(* Logix 5000 project; controller reports 1756-L63 rev 20.15; software revision 20.04; part 16 of 52 *)

        [783].log_data[6].valid := 1, [783].log_data[7].valid := 1, [783].log_data[8].valid := 1, [783].log_data[9].valid := 1, [783].log_data[10].valid := 1, [783].log_data[11].valid := 1, [783].log_data[12].valid := 1, [783].log_data[13].valid := 1, [783].log_data[14].valid := 1, [783].log_data[15].valid := 1, [783].log_data[16].valid := 1, [783].log_data[17].valid := 1, [783].log_data[18].valid := 1, [783].log_data[19].valid := 1, [783].time.Year := 2023, [783].time.Month := 1, [783].time.Day := 12, [783].time.Hour := 9, [783].time.Minute := 39, [783].time.Second := 59, [784].log_data[0].min := 1.0, [784].log_data[0].max := 1.0, [784].log_data[0].total := 300.0, [784].log_data[0].time := 300.0, [784].log_data[0].minminute := 40, [784].log_data[0].maxminute := 40, [784].log_data[0].valid := 1, [784].log_data[1].valid := 1, [784].log_data[2].valid := 1, [784].log_data[3].valid := 1, [784].log_data[4].valid := 1, [784].log_data[5].valid := 1, [784].log_data[6].valid := 1, [784].log_data[7].valid := 1, [784].log_data[8].valid := 1, [784].log_data[9].valid := 1, [784].log_data[10].valid := 1, [784].log_data[11].valid := 1, [784].log_data[12].valid := 1, [784].log_data[13].valid := 1, [784].log_data[14].valid := 1, [784].log_data[15].valid := 1, [784].log_data[16].valid := 1, [784].log_data[17].valid := 1, [784].log_data[18].valid := 1, [784].log_data[19].valid := 1, [784].time.Year := 2023, [784].time.Month := 1, [784].time.Day := 12, [784].time.Hour := 9, [784].time.Minute := 44, [784].time.Second := 59, [785].log_data[0].min := 1.0, [785].log_data[0].max := 1.0, [785].log_data[0].total := 300.0, [785].log_data[0].time := 300.0, [785].log_data[0].minminute := 45, [785].log_data[0].maxminute := 45, [785].log_data[0].valid := 1, [785].log_data[1].valid := 1,
        [785].log_data[2].valid := 1, [785].log_data[3].valid := 1, [785].log_data[4].valid := 1, [785].log_data[5].valid := 1, [785].log_data[6].valid := 1, [785].log_data[7].valid := 1, [785].log_data[8].valid := 1, [785].log_data[9].valid := 1, [785].log_data[10].valid := 1, [785].log_data[11].valid := 1, [785].log_data[12].valid := 1, [785].log_data[13].valid := 1, [785].log_data[14].valid := 1, [785].log_data[15].valid := 1, [785].log_data[16].valid := 1, [785].log_data[17].valid := 1, [785].log_data[18].valid := 1, [785].log_data[19].valid := 1, [785].time.Year := 2023, [785].time.Month := 1, [785].time.Day := 12, [785].time.Hour := 9, [785].time.Minute := 49, [785].time.Second := 59, [786].log_data[0].min := 1.0, [786].log_data[0].max := 1.0, [786].log_data[0].total := 300.0, [786].log_data[0].time := 300.0, [786].log_data[0].minminute := 50, [786].log_data[0].maxminute := 50, [786].log_data[0].valid := 1, [786].log_data[1].valid := 1, [786].log_data[2].valid := 1, [786].log_data[3].valid := 1, [786].log_data[4].valid := 1, [786].log_data[5].valid := 1, [786].log_data[6].valid := 1, [786].log_data[7].valid := 1, [786].log_data[8].valid := 1, [786].log_data[9].valid := 1, [786].log_data[10].valid := 1, [786].log_data[11].valid := 1, [786].log_data[12].valid := 1, [786].log_data[13].valid := 1, [786].log_data[14].valid := 1, [786].log_data[15].valid := 1, [786].log_data[16].valid := 1, [786].log_data[17].valid := 1, [786].log_data[18].valid := 1, [786].log_data[19].valid := 1, [786].time.Year := 2023, [786].time.Month := 1, [786].time.Day := 12, [786].time.Hour := 9, [786].time.Minute := 54, [786].time.Second := 59, [787].log_data[0].min := 1.0, [787].log_data[0].max := 1.0, [787].log_data[0].total := 300.0, [787].log_data[0].time := 300.0,
        [787].log_data[0].minminute := 55, [787].log_data[0].maxminute := 55, [787].log_data[0].valid := 1, [787].log_data[1].valid := 1, [787].log_data[2].valid := 1, [787].log_data[3].valid := 1, [787].log_data[4].valid := 1, [787].log_data[5].valid := 1, [787].log_data[6].valid := 1, [787].log_data[7].valid := 1, [787].log_data[8].valid := 1, [787].log_data[9].valid := 1, [787].log_data[10].valid := 1, [787].log_data[11].valid := 1, [787].log_data[12].valid := 1, [787].log_data[13].valid := 1, [787].log_data[14].valid := 1, [787].log_data[15].valid := 1, [787].log_data[16].valid := 1, [787].log_data[17].valid := 1, [787].log_data[18].valid := 1, [787].log_data[19].valid := 1, [787].time.Year := 2023, [787].time.Month := 1, [787].time.Day := 12, [787].time.Hour := 9, [787].time.Minute := 59, [787].time.Second := 59, [788].log_data[0].min := 1.0, [788].log_data[0].max := 1.0, [788].log_data[0].total := 300.0, [788].log_data[0].time := 300.0, [788].log_data[0].valid := 1, [788].log_data[1].valid := 1, [788].log_data[2].valid := 1, [788].log_data[3].valid := 1, [788].log_data[4].valid := 1, [788].log_data[5].valid := 1, [788].log_data[6].valid := 1, [788].log_data[7].valid := 1, [788].log_data[8].valid := 1, [788].log_data[9].valid := 1, [788].log_data[10].valid := 1, [788].log_data[11].valid := 1, [788].log_data[12].valid := 1, [788].log_data[13].valid := 1, [788].log_data[14].valid := 1, [788].log_data[15].valid := 1, [788].log_data[16].valid := 1, [788].log_data[17].valid := 1, [788].log_data[18].valid := 1, [788].log_data[19].valid := 1, [788].time.Year := 2023, [788].time.Month := 1, [788].time.Day := 12, [788].time.Hour := 10, [788].time.Minute := 4, [788].time.Second := 59, [789].log_data[0].min := 1.0, [789].log_data[0].max := 1.0,
        [789].log_data[0].total := 300.0, [789].log_data[0].time := 300.0, [789].log_data[0].minminute := 5, [789].log_data[0].maxminute := 5, [789].log_data[0].valid := 1, [789].log_data[1].valid := 1, [789].log_data[2].valid := 1, [789].log_data[3].valid := 1, [789].log_data[4].valid := 1, [789].log_data[5].valid := 1, [789].log_data[6].valid := 1, [789].log_data[7].valid := 1, [789].log_data[8].valid := 1, [789].log_data[9].valid := 1, [789].log_data[10].valid := 1, [789].log_data[11].valid := 1, [789].log_data[12].valid := 1, [789].log_data[13].valid := 1, [789].log_data[14].valid := 1, [789].log_data[15].valid := 1, [789].log_data[16].valid := 1, [789].log_data[17].valid := 1, [789].log_data[18].valid := 1, [789].log_data[19].valid := 1, [789].time.Year := 2023, [789].time.Month := 1, [789].time.Day := 12, [789].time.Hour := 10, [789].time.Minute := 9, [789].time.Second := 59, [790].log_data[0].min := 1.0, [790].log_data[0].max := 1.0, [790].log_data[0].total := 300.0, [790].log_data[0].time := 300.0, [790].log_data[0].minminute := 10, [790].log_data[0].maxminute := 10, [790].log_data[0].valid := 1, [790].log_data[1].valid := 1, [790].log_data[2].valid := 1, [790].log_data[3].valid := 1, [790].log_data[4].valid := 1, [790].log_data[5].valid := 1, [790].log_data[6].valid := 1, [790].log_data[7].valid := 1, [790].log_data[8].valid := 1, [790].log_data[9].valid := 1, [790].log_data[10].valid := 1, [790].log_data[11].valid := 1, [790].log_data[12].valid := 1, [790].log_data[13].valid := 1, [790].log_data[14].valid := 1, [790].log_data[15].valid := 1, [790].log_data[16].valid := 1, [790].log_data[17].valid := 1, [790].log_data[18].valid := 1, [790].log_data[19].valid := 1, [790].time.Year := 2023, [790].time.Month := 1, [790].time.Day := 12, [790].time.Hour := 10,
        [790].time.Minute := 14, [790].time.Second := 59, [791].log_data[0].min := 1.0, [791].log_data[0].max := 1.0, [791].log_data[0].total := 300.0, [791].log_data[0].time := 300.0, [791].log_data[0].minminute := 15, [791].log_data[0].maxminute := 15, [791].log_data[0].valid := 1, [791].log_data[1].valid := 1, [791].log_data[2].valid := 1, [791].log_data[3].valid := 1, [791].log_data[4].valid := 1, [791].log_data[5].valid := 1, [791].log_data[6].valid := 1, [791].log_data[7].valid := 1, [791].log_data[8].valid := 1, [791].log_data[9].valid := 1, [791].log_data[10].valid := 1, [791].log_data[11].valid := 1, [791].log_data[12].valid := 1, [791].log_data[13].valid := 1, [791].log_data[14].valid := 1, [791].log_data[15].valid := 1, [791].log_data[16].valid := 1, [791].log_data[17].valid := 1, [791].log_data[18].valid := 1, [791].log_data[19].valid := 1, [791].time.Year := 2023, [791].time.Month := 1, [791].time.Day := 12, [791].time.Hour := 10, [791].time.Minute := 19, [791].time.Second := 59, [792].log_data[0].min := 1.0, [792].log_data[0].max := 1.0, [792].log_data[0].total := 300.0, [792].log_data[0].time := 300.0, [792].log_data[0].minminute := 20, [792].log_data[0].maxminute := 20, [792].log_data[0].valid := 1, [792].log_data[1].valid := 1, [792].log_data[2].valid := 1, [792].log_data[3].valid := 1, [792].log_data[4].valid := 1, [792].log_data[5].valid := 1, [792].log_data[6].valid := 1, [792].log_data[7].valid := 1, [792].log_data[8].valid := 1, [792].log_data[9].valid := 1, [792].log_data[10].valid := 1, [792].log_data[11].valid := 1, [792].log_data[12].valid := 1, [792].log_data[13].valid := 1, [792].log_data[14].valid := 1, [792].log_data[15].valid := 1, [792].log_data[16].valid := 1, [792].log_data[17].valid := 1, [792].log_data[18].valid := 1, [792].log_data[19].valid := 1,
        [792].time.Year := 2023, [792].time.Month := 1, [792].time.Day := 12, [792].time.Hour := 10, [792].time.Minute := 24, [792].time.Second := 59, [793].log_data[0].min := 1.0, [793].log_data[0].max := 1.0, [793].log_data[0].total := 300.0, [793].log_data[0].time := 300.0, [793].log_data[0].minminute := 25, [793].log_data[0].maxminute := 25, [793].log_data[0].valid := 1, [793].log_data[1].valid := 1, [793].log_data[2].valid := 1, [793].log_data[3].valid := 1, [793].log_data[4].valid := 1, [793].log_data[5].valid := 1, [793].log_data[6].valid := 1, [793].log_data[7].valid := 1, [793].log_data[8].valid := 1, [793].log_data[9].valid := 1, [793].log_data[10].valid := 1, [793].log_data[11].valid := 1, [793].log_data[12].valid := 1, [793].log_data[13].valid := 1, [793].log_data[14].valid := 1, [793].log_data[15].valid := 1, [793].log_data[16].valid := 1, [793].log_data[17].valid := 1, [793].log_data[18].valid := 1, [793].log_data[19].valid := 1, [793].time.Year := 2023, [793].time.Month := 1, [793].time.Day := 12, [793].time.Hour := 10, [793].time.Minute := 29, [793].time.Second := 59, [794].log_data[0].min := 1.0, [794].log_data[0].max := 1.0, [794].log_data[0].total := 300.0, [794].log_data[0].time := 300.0, [794].log_data[0].minminute := 30, [794].log_data[0].maxminute := 30, [794].log_data[0].valid := 1, [794].log_data[1].valid := 1, [794].log_data[2].valid := 1, [794].log_data[3].valid := 1, [794].log_data[4].valid := 1, [794].log_data[5].valid := 1, [794].log_data[6].valid := 1, [794].log_data[7].valid := 1, [794].log_data[8].valid := 1, [794].log_data[9].valid := 1, [794].log_data[10].valid := 1, [794].log_data[11].valid := 1, [794].log_data[12].valid := 1, [794].log_data[13].valid := 1, [794].log_data[14].valid := 1, [794].log_data[15].valid := 1,
        [794].log_data[16].valid := 1, [794].log_data[17].valid := 1, [794].log_data[18].valid := 1, [794].log_data[19].valid := 1, [794].time.Year := 2023, [794].time.Month := 1, [794].time.Day := 12, [794].time.Hour := 10, [794].time.Minute := 34, [794].time.Second := 59, [795].log_data[0].min := 1.0, [795].log_data[0].max := 1.0, [795].log_data[0].total := 300.0, [795].log_data[0].time := 300.0, [795].log_data[0].minminute := 35, [795].log_data[0].maxminute := 35, [795].log_data[0].valid := 1, [795].log_data[1].valid := 1, [795].log_data[2].valid := 1, [795].log_data[3].valid := 1, [795].log_data[4].valid := 1, [795].log_data[5].valid := 1, [795].log_data[6].valid := 1, [795].log_data[7].valid := 1, [795].log_data[8].valid := 1, [795].log_data[9].valid := 1, [795].log_data[10].valid := 1, [795].log_data[11].valid := 1, [795].log_data[12].valid := 1, [795].log_data[13].valid := 1, [795].log_data[14].valid := 1, [795].log_data[15].valid := 1, [795].log_data[16].valid := 1, [795].log_data[17].valid := 1, [795].log_data[18].valid := 1, [795].log_data[19].valid := 1, [795].time.Year := 2023, [795].time.Month := 1, [795].time.Day := 12, [795].time.Hour := 10, [795].time.Minute := 39, [795].time.Second := 59, [796].log_data[0].min := 1.0, [796].log_data[0].max := 1.0, [796].log_data[0].total := 300.0, [796].log_data[0].time := 300.0, [796].log_data[0].minminute := 40, [796].log_data[0].maxminute := 40, [796].log_data[0].valid := 1, [796].log_data[1].valid := 1, [796].log_data[2].valid := 1, [796].log_data[3].valid := 1, [796].log_data[4].valid := 1, [796].log_data[5].valid := 1, [796].log_data[6].valid := 1, [796].log_data[7].valid := 1, [796].log_data[8].valid := 1, [796].log_data[9].valid := 1, [796].log_data[10].valid := 1, [796].log_data[11].valid := 1,
        [796].log_data[12].valid := 1, [796].log_data[13].valid := 1, [796].log_data[14].valid := 1, [796].log_data[15].valid := 1, [796].log_data[16].valid := 1, [796].log_data[17].valid := 1, [796].log_data[18].valid := 1, [796].log_data[19].valid := 1, [796].time.Year := 2023, [796].time.Month := 1, [796].time.Day := 12, [796].time.Hour := 10, [796].time.Minute := 44, [796].time.Second := 59, [797].log_data[0].min := 1.0, [797].log_data[0].max := 1.0, [797].log_data[0].total := 300.0, [797].log_data[0].time := 300.0, [797].log_data[0].minminute := 45, [797].log_data[0].maxminute := 45, [797].log_data[0].valid := 1, [797].log_data[1].valid := 1, [797].log_data[2].valid := 1, [797].log_data[3].valid := 1, [797].log_data[4].valid := 1, [797].log_data[5].valid := 1, [797].log_data[6].valid := 1, [797].log_data[7].valid := 1, [797].log_data[8].valid := 1, [797].log_data[9].valid := 1, [797].log_data[10].valid := 1, [797].log_data[11].valid := 1, [797].log_data[12].valid := 1, [797].log_data[13].valid := 1, [797].log_data[14].valid := 1, [797].log_data[15].valid := 1, [797].log_data[16].valid := 1, [797].log_data[17].valid := 1, [797].log_data[18].valid := 1, [797].log_data[19].valid := 1, [797].time.Year := 2023, [797].time.Month := 1, [797].time.Day := 12, [797].time.Hour := 10, [797].time.Minute := 49, [797].time.Second := 59, [798].log_data[0].min := 1.0, [798].log_data[0].max := 1.0, [798].log_data[0].total := 300.0, [798].log_data[0].time := 300.0, [798].log_data[0].minminute := 50, [798].log_data[0].maxminute := 50, [798].log_data[0].valid := 1, [798].log_data[1].valid := 1, [798].log_data[2].valid := 1, [798].log_data[3].valid := 1, [798].log_data[4].valid := 1, [798].log_data[5].valid := 1, [798].log_data[6].valid := 1, [798].log_data[7].valid := 1,
        [798].log_data[8].valid := 1, [798].log_data[9].valid := 1, [798].log_data[10].valid := 1, [798].log_data[11].valid := 1, [798].log_data[12].valid := 1, [798].log_data[13].valid := 1, [798].log_data[14].valid := 1, [798].log_data[15].valid := 1, [798].log_data[16].valid := 1, [798].log_data[17].valid := 1, [798].log_data[18].valid := 1, [798].log_data[19].valid := 1, [798].time.Year := 2023, [798].time.Month := 1, [798].time.Day := 12, [798].time.Hour := 10, [798].time.Minute := 54, [798].time.Second := 59, [799].log_data[0].min := 1.0, [799].log_data[0].max := 1.0, [799].log_data[0].total := 300.0, [799].log_data[0].time := 300.0, [799].log_data[0].minminute := 55, [799].log_data[0].maxminute := 55, [799].log_data[0].valid := 1, [799].log_data[1].valid := 1, [799].log_data[2].valid := 1, [799].log_data[3].valid := 1, [799].log_data[4].valid := 1, [799].log_data[5].valid := 1, [799].log_data[6].valid := 1, [799].log_data[7].valid := 1, [799].log_data[8].valid := 1, [799].log_data[9].valid := 1, [799].log_data[10].valid := 1, [799].log_data[11].valid := 1, [799].log_data[12].valid := 1, [799].log_data[13].valid := 1, [799].log_data[14].valid := 1, [799].log_data[15].valid := 1, [799].log_data[16].valid := 1, [799].log_data[17].valid := 1, [799].log_data[18].valid := 1, [799].log_data[19].valid := 1, [799].time.Year := 2023, [799].time.Month := 1, [799].time.Day := 12, [799].time.Hour := 10, [799].time.Minute := 59, [799].time.Second := 59, [800].log_data[0].min := 1.0, [800].log_data[0].max := 1.0, [800].log_data[0].total := 300.0, [800].log_data[0].time := 300.0, [800].log_data[0].valid := 1, [800].log_data[1].valid := 1, [800].log_data[2].valid := 1, [800].log_data[3].valid := 1, [800].log_data[4].valid := 1, [800].log_data[5].valid := 1,
        [800].log_data[6].valid := 1, [800].log_data[7].valid := 1, [800].log_data[8].valid := 1, [800].log_data[9].valid := 1, [800].log_data[10].valid := 1, [800].log_data[11].valid := 1, [800].log_data[12].valid := 1, [800].log_data[13].valid := 1, [800].log_data[14].valid := 1, [800].log_data[15].valid := 1, [800].log_data[16].valid := 1, [800].log_data[17].valid := 1, [800].log_data[18].valid := 1, [800].log_data[19].valid := 1, [800].time.Year := 2023, [800].time.Month := 1, [800].time.Day := 12, [800].time.Hour := 11, [800].time.Minute := 4, [800].time.Second := 59, [801].log_data[0].min := 1.0, [801].log_data[0].max := 1.0, [801].log_data[0].total := 300.0, [801].log_data[0].time := 300.0, [801].log_data[0].minminute := 5, [801].log_data[0].maxminute := 5, [801].log_data[0].valid := 1, [801].log_data[1].valid := 1, [801].log_data[2].valid := 1, [801].log_data[3].valid := 1, [801].log_data[4].valid := 1, [801].log_data[5].valid := 1, [801].log_data[6].valid := 1, [801].log_data[7].valid := 1, [801].log_data[8].valid := 1, [801].log_data[9].valid := 1, [801].log_data[10].valid := 1, [801].log_data[11].valid := 1, [801].log_data[12].valid := 1, [801].log_data[13].valid := 1, [801].log_data[14].valid := 1, [801].log_data[15].valid := 1, [801].log_data[16].valid := 1, [801].log_data[17].valid := 1, [801].log_data[18].valid := 1, [801].log_data[19].valid := 1, [801].time.Year := 2023, [801].time.Month := 1, [801].time.Day := 12, [801].time.Hour := 11, [801].time.Minute := 9, [801].time.Second := 59, [802].log_data[0].min := 1.0, [802].log_data[0].max := 1.0, [802].log_data[0].total := 300.0, [802].log_data[0].time := 300.0, [802].log_data[0].minminute := 10, [802].log_data[0].maxminute := 10, [802].log_data[0].valid := 1, [802].log_data[1].valid := 1,
        [802].log_data[2].valid := 1, [802].log_data[3].valid := 1, [802].log_data[4].valid := 1, [802].log_data[5].valid := 1, [802].log_data[6].valid := 1, [802].log_data[7].valid := 1, [802].log_data[8].valid := 1, [802].log_data[9].valid := 1, [802].log_data[10].valid := 1, [802].log_data[11].valid := 1, [802].log_data[12].valid := 1, [802].log_data[13].valid := 1, [802].log_data[14].valid := 1, [802].log_data[15].valid := 1, [802].log_data[16].valid := 1, [802].log_data[17].valid := 1, [802].log_data[18].valid := 1, [802].log_data[19].valid := 1, [802].time.Year := 2023, [802].time.Month := 1, [802].time.Day := 12, [802].time.Hour := 11, [802].time.Minute := 14, [802].time.Second := 59, [803].log_data[0].min := 1.0, [803].log_data[0].max := 1.0, [803].log_data[0].total := 300.0, [803].log_data[0].time := 300.0, [803].log_data[0].minminute := 15, [803].log_data[0].maxminute := 15, [803].log_data[0].valid := 1, [803].log_data[1].valid := 1, [803].log_data[2].valid := 1, [803].log_data[3].valid := 1, [803].log_data[4].valid := 1, [803].log_data[5].valid := 1, [803].log_data[6].valid := 1, [803].log_data[7].valid := 1, [803].log_data[8].valid := 1, [803].log_data[9].valid := 1, [803].log_data[10].valid := 1, [803].log_data[11].valid := 1, [803].log_data[12].valid := 1, [803].log_data[13].valid := 1, [803].log_data[14].valid := 1, [803].log_data[15].valid := 1, [803].log_data[16].valid := 1, [803].log_data[17].valid := 1, [803].log_data[18].valid := 1, [803].log_data[19].valid := 1, [803].time.Year := 2023, [803].time.Month := 1, [803].time.Day := 12, [803].time.Hour := 11, [803].time.Minute := 19, [803].time.Second := 59, [804].log_data[0].min := 1.0, [804].log_data[0].max := 1.0, [804].log_data[0].total := 300.0, [804].log_data[0].time := 300.0,
        [804].log_data[0].minminute := 20, [804].log_data[0].maxminute := 20, [804].log_data[0].valid := 1, [804].log_data[1].valid := 1, [804].log_data[2].valid := 1, [804].log_data[3].valid := 1, [804].log_data[4].valid := 1, [804].log_data[5].valid := 1, [804].log_data[6].valid := 1, [804].log_data[7].valid := 1, [804].log_data[8].valid := 1, [804].log_data[9].valid := 1, [804].log_data[10].valid := 1, [804].log_data[11].valid := 1, [804].log_data[12].valid := 1, [804].log_data[13].valid := 1, [804].log_data[14].valid := 1, [804].log_data[15].valid := 1, [804].log_data[16].valid := 1, [804].log_data[17].valid := 1, [804].log_data[18].valid := 1, [804].log_data[19].valid := 1, [804].time.Year := 2023, [804].time.Month := 1, [804].time.Day := 12, [804].time.Hour := 11, [804].time.Minute := 24, [804].time.Second := 59, [805].log_data[0].min := 1.0, [805].log_data[0].max := 1.0, [805].log_data[0].total := 300.0, [805].log_data[0].time := 300.0, [805].log_data[0].minminute := 25, [805].log_data[0].maxminute := 25, [805].log_data[0].valid := 1, [805].log_data[1].valid := 1, [805].log_data[2].valid := 1, [805].log_data[3].valid := 1, [805].log_data[4].valid := 1, [805].log_data[5].valid := 1, [805].log_data[6].valid := 1, [805].log_data[7].valid := 1, [805].log_data[8].valid := 1, [805].log_data[9].valid := 1, [805].log_data[10].valid := 1, [805].log_data[11].valid := 1, [805].log_data[12].valid := 1, [805].log_data[13].valid := 1, [805].log_data[14].valid := 1, [805].log_data[15].valid := 1, [805].log_data[16].valid := 1, [805].log_data[17].valid := 1, [805].log_data[18].valid := 1, [805].log_data[19].valid := 1, [805].time.Year := 2023, [805].time.Month := 1, [805].time.Day := 12, [805].time.Hour := 11, [805].time.Minute := 29, [805].time.Second := 59,
        [806].log_data[0].min := 1.0, [806].log_data[0].max := 1.0, [806].log_data[0].total := 300.0, [806].log_data[0].time := 300.0, [806].log_data[0].minminute := 30, [806].log_data[0].maxminute := 30, [806].log_data[0].valid := 1, [806].log_data[1].valid := 1, [806].log_data[2].valid := 1, [806].log_data[3].valid := 1, [806].log_data[4].valid := 1, [806].log_data[5].valid := 1, [806].log_data[6].valid := 1, [806].log_data[7].valid := 1, [806].log_data[8].valid := 1, [806].log_data[9].valid := 1, [806].log_data[10].valid := 1, [806].log_data[11].valid := 1, [806].log_data[12].valid := 1, [806].log_data[13].valid := 1, [806].log_data[14].valid := 1, [806].log_data[15].valid := 1, [806].log_data[16].valid := 1, [806].log_data[17].valid := 1, [806].log_data[18].valid := 1, [806].log_data[19].valid := 1, [806].time.Year := 2023, [806].time.Month := 1, [806].time.Day := 12, [806].time.Hour := 11, [806].time.Minute := 34, [806].time.Second := 59, [807].log_data[0].min := 1.0, [807].log_data[0].max := 1.0, [807].log_data[0].total := 300.0, [807].log_data[0].time := 300.0, [807].log_data[0].minminute := 35, [807].log_data[0].maxminute := 35, [807].log_data[0].valid := 1, [807].log_data[1].valid := 1, [807].log_data[2].valid := 1, [807].log_data[3].valid := 1, [807].log_data[4].valid := 1, [807].log_data[5].valid := 1, [807].log_data[6].valid := 1, [807].log_data[7].valid := 1, [807].log_data[8].valid := 1, [807].log_data[9].valid := 1, [807].log_data[10].valid := 1, [807].log_data[11].valid := 1, [807].log_data[12].valid := 1, [807].log_data[13].valid := 1, [807].log_data[14].valid := 1, [807].log_data[15].valid := 1, [807].log_data[16].valid := 1, [807].log_data[17].valid := 1, [807].log_data[18].valid := 1, [807].log_data[19].valid := 1, [807].time.Year := 2023, [807].time.Month := 1,
        [807].time.Day := 12, [807].time.Hour := 11, [807].time.Minute := 39, [807].time.Second := 59, [808].log_data[0].min := 1.0, [808].log_data[0].max := 1.0, [808].log_data[0].total := 300.0, [808].log_data[0].time := 300.0, [808].log_data[0].minminute := 40, [808].log_data[0].maxminute := 40, [808].log_data[0].valid := 1, [808].log_data[1].valid := 1, [808].log_data[2].valid := 1, [808].log_data[3].valid := 1, [808].log_data[4].valid := 1, [808].log_data[5].valid := 1, [808].log_data[6].valid := 1, [808].log_data[7].valid := 1, [808].log_data[8].valid := 1, [808].log_data[9].valid := 1, [808].log_data[10].valid := 1, [808].log_data[11].valid := 1, [808].log_data[12].valid := 1, [808].log_data[13].valid := 1, [808].log_data[14].valid := 1, [808].log_data[15].valid := 1, [808].log_data[16].valid := 1, [808].log_data[17].valid := 1, [808].log_data[18].valid := 1, [808].log_data[19].valid := 1, [808].time.Year := 2023, [808].time.Month := 1, [808].time.Day := 12, [808].time.Hour := 11, [808].time.Minute := 44, [808].time.Second := 59, [809].log_data[0].min := 1.0, [809].log_data[0].max := 1.0, [809].log_data[0].total := 300.0, [809].log_data[0].time := 300.0, [809].log_data[0].minminute := 45, [809].log_data[0].maxminute := 45, [809].log_data[0].valid := 1, [809].log_data[1].valid := 1, [809].log_data[2].valid := 1, [809].log_data[3].valid := 1, [809].log_data[4].valid := 1, [809].log_data[5].valid := 1, [809].log_data[6].valid := 1, [809].log_data[7].valid := 1, [809].log_data[8].valid := 1, [809].log_data[9].valid := 1, [809].log_data[10].valid := 1, [809].log_data[11].valid := 1, [809].log_data[12].valid := 1, [809].log_data[13].valid := 1, [809].log_data[14].valid := 1, [809].log_data[15].valid := 1, [809].log_data[16].valid := 1, [809].log_data[17].valid := 1,
        [809].log_data[18].valid := 1, [809].log_data[19].valid := 1, [809].time.Year := 2023, [809].time.Month := 1, [809].time.Day := 12, [809].time.Hour := 11, [809].time.Minute := 49, [809].time.Second := 59, [810].log_data[0].min := 1.0, [810].log_data[0].max := 1.0, [810].log_data[0].total := 300.0, [810].log_data[0].time := 300.0, [810].log_data[0].minminute := 50, [810].log_data[0].maxminute := 50, [810].log_data[0].valid := 1, [810].log_data[1].valid := 1, [810].log_data[2].valid := 1, [810].log_data[3].valid := 1, [810].log_data[4].valid := 1, [810].log_data[5].valid := 1, [810].log_data[6].valid := 1, [810].log_data[7].valid := 1, [810].log_data[8].valid := 1, [810].log_data[9].valid := 1, [810].log_data[10].valid := 1, [810].log_data[11].valid := 1, [810].log_data[12].valid := 1, [810].log_data[13].valid := 1, [810].log_data[14].valid := 1, [810].log_data[15].valid := 1, [810].log_data[16].valid := 1, [810].log_data[17].valid := 1, [810].log_data[18].valid := 1, [810].log_data[19].valid := 1, [810].time.Year := 2023, [810].time.Month := 1, [810].time.Day := 12, [810].time.Hour := 11, [810].time.Minute := 54, [810].time.Second := 59, [811].log_data[0].min := 1.0, [811].log_data[0].max := 1.0, [811].log_data[0].total := 300.0, [811].log_data[0].time := 300.0, [811].log_data[0].minminute := 55, [811].log_data[0].maxminute := 55, [811].log_data[0].valid := 1, [811].log_data[1].valid := 1, [811].log_data[2].valid := 1, [811].log_data[3].valid := 1, [811].log_data[4].valid := 1, [811].log_data[5].valid := 1, [811].log_data[6].valid := 1, [811].log_data[7].valid := 1, [811].log_data[8].valid := 1, [811].log_data[9].valid := 1, [811].log_data[10].valid := 1, [811].log_data[11].valid := 1, [811].log_data[12].valid := 1, [811].log_data[13].valid := 1,
        [811].log_data[14].valid := 1, [811].log_data[15].valid := 1, [811].log_data[16].valid := 1, [811].log_data[17].valid := 1, [811].log_data[18].valid := 1, [811].log_data[19].valid := 1, [811].time.Year := 2023, [811].time.Month := 1, [811].time.Day := 12, [811].time.Hour := 11, [811].time.Minute := 59, [811].time.Second := 59, [812].log_data[0].min := 1.0, [812].log_data[0].max := 1.0, [812].log_data[0].total := 300.0, [812].log_data[0].time := 300.0, [812].log_data[0].valid := 1, [812].log_data[1].valid := 1, [812].log_data[2].valid := 1, [812].log_data[3].valid := 1, [812].log_data[4].valid := 1, [812].log_data[5].valid := 1, [812].log_data[6].valid := 1, [812].log_data[7].valid := 1, [812].log_data[8].valid := 1, [812].log_data[9].valid := 1, [812].log_data[10].valid := 1, [812].log_data[11].valid := 1, [812].log_data[12].valid := 1, [812].log_data[13].valid := 1, [812].log_data[14].valid := 1, [812].log_data[15].valid := 1, [812].log_data[16].valid := 1, [812].log_data[17].valid := 1, [812].log_data[18].valid := 1, [812].log_data[19].valid := 1, [812].time.Year := 2023, [812].time.Month := 1, [812].time.Day := 12, [812].time.Hour := 12, [812].time.Minute := 4, [812].time.Second := 59, [813].log_data[0].min := 1.0, [813].log_data[0].max := 1.0, [813].log_data[0].total := 300.0, [813].log_data[0].time := 300.0, [813].log_data[0].minminute := 5, [813].log_data[0].maxminute := 5, [813].log_data[0].valid := 1, [813].log_data[1].valid := 1, [813].log_data[2].valid := 1, [813].log_data[3].valid := 1, [813].log_data[4].valid := 1, [813].log_data[5].valid := 1, [813].log_data[6].valid := 1, [813].log_data[7].valid := 1, [813].log_data[8].valid := 1, [813].log_data[9].valid := 1, [813].log_data[10].valid := 1, [813].log_data[11].valid := 1,
        [813].log_data[12].valid := 1, [813].log_data[13].valid := 1, [813].log_data[14].valid := 1, [813].log_data[15].valid := 1, [813].log_data[16].valid := 1, [813].log_data[17].valid := 1, [813].log_data[18].valid := 1, [813].log_data[19].valid := 1, [813].time.Year := 2023, [813].time.Month := 1, [813].time.Day := 12, [813].time.Hour := 12, [813].time.Minute := 9, [813].time.Second := 59, [814].log_data[0].min := 1.0, [814].log_data[0].max := 1.0, [814].log_data[0].total := 300.0, [814].log_data[0].time := 300.0, [814].log_data[0].minminute := 10, [814].log_data[0].maxminute := 10, [814].log_data[0].valid := 1, [814].log_data[1].valid := 1, [814].log_data[2].valid := 1, [814].log_data[3].valid := 1, [814].log_data[4].valid := 1, [814].log_data[5].valid := 1, [814].log_data[6].valid := 1, [814].log_data[7].valid := 1, [814].log_data[8].valid := 1, [814].log_data[9].valid := 1, [814].log_data[10].valid := 1, [814].log_data[11].valid := 1, [814].log_data[12].valid := 1, [814].log_data[13].valid := 1, [814].log_data[14].valid := 1, [814].log_data[15].valid := 1, [814].log_data[16].valid := 1, [814].log_data[17].valid := 1, [814].log_data[18].valid := 1, [814].log_data[19].valid := 1, [814].time.Year := 2023, [814].time.Month := 1, [814].time.Day := 12, [814].time.Hour := 12, [814].time.Minute := 14, [814].time.Second := 59, [815].log_data[0].min := 1.0, [815].log_data[0].max := 1.0, [815].log_data[0].total := 300.0, [815].log_data[0].time := 300.0, [815].log_data[0].minminute := 15, [815].log_data[0].maxminute := 15, [815].log_data[0].valid := 1, [815].log_data[1].valid := 1, [815].log_data[2].valid := 1, [815].log_data[3].valid := 1, [815].log_data[4].valid := 1, [815].log_data[5].valid := 1, [815].log_data[6].valid := 1, [815].log_data[7].valid := 1,
        [815].log_data[8].valid := 1, [815].log_data[9].valid := 1, [815].log_data[10].valid := 1, [815].log_data[11].valid := 1, [815].log_data[12].valid := 1, [815].log_data[13].valid := 1, [815].log_data[14].valid := 1, [815].log_data[15].valid := 1, [815].log_data[16].valid := 1, [815].log_data[17].valid := 1, [815].log_data[18].valid := 1, [815].log_data[19].valid := 1, [815].time.Year := 2023, [815].time.Month := 1, [815].time.Day := 12, [815].time.Hour := 12, [815].time.Minute := 19, [815].time.Second := 59, [816].log_data[0].min := 1.0, [816].log_data[0].max := 1.0, [816].log_data[0].total := 300.0, [816].log_data[0].time := 300.0, [816].log_data[0].minminute := 20, [816].log_data[0].maxminute := 20, [816].log_data[0].valid := 1, [816].log_data[1].valid := 1, [816].log_data[2].valid := 1, [816].log_data[3].valid := 1, [816].log_data[4].valid := 1, [816].log_data[5].valid := 1, [816].log_data[6].valid := 1, [816].log_data[7].valid := 1, [816].log_data[8].valid := 1, [816].log_data[9].valid := 1, [816].log_data[10].valid := 1, [816].log_data[11].valid := 1, [816].log_data[12].valid := 1, [816].log_data[13].valid := 1, [816].log_data[14].valid := 1, [816].log_data[15].valid := 1, [816].log_data[16].valid := 1, [816].log_data[17].valid := 1, [816].log_data[18].valid := 1, [816].log_data[19].valid := 1, [816].time.Year := 2023, [816].time.Month := 1, [816].time.Day := 12, [816].time.Hour := 12, [816].time.Minute := 24, [816].time.Second := 59, [817].log_data[0].min := 1.0, [817].log_data[0].max := 1.0, [817].log_data[0].total := 300.0, [817].log_data[0].time := 300.0, [817].log_data[0].minminute := 25, [817].log_data[0].maxminute := 25, [817].log_data[0].valid := 1, [817].log_data[1].valid := 1, [817].log_data[2].valid := 1, [817].log_data[3].valid := 1,
        [817].log_data[4].valid := 1, [817].log_data[5].valid := 1, [817].log_data[6].valid := 1, [817].log_data[7].valid := 1, [817].log_data[8].valid := 1, [817].log_data[9].valid := 1, [817].log_data[10].valid := 1, [817].log_data[11].valid := 1, [817].log_data[12].valid := 1, [817].log_data[13].valid := 1, [817].log_data[14].valid := 1, [817].log_data[15].valid := 1, [817].log_data[16].valid := 1, [817].log_data[17].valid := 1, [817].log_data[18].valid := 1, [817].log_data[19].valid := 1, [817].time.Year := 2023, [817].time.Month := 1, [817].time.Day := 12, [817].time.Hour := 12, [817].time.Minute := 29, [817].time.Second := 59, [818].log_data[0].min := 1.0, [818].log_data[0].max := 1.0, [818].log_data[0].total := 300.0, [818].log_data[0].time := 300.0, [818].log_data[0].minminute := 30, [818].log_data[0].maxminute := 30, [818].log_data[0].valid := 1, [818].log_data[1].valid := 1, [818].log_data[2].valid := 1, [818].log_data[3].valid := 1, [818].log_data[4].valid := 1, [818].log_data[5].valid := 1, [818].log_data[6].valid := 1, [818].log_data[7].valid := 1, [818].log_data[8].valid := 1, [818].log_data[9].valid := 1, [818].log_data[10].valid := 1, [818].log_data[11].valid := 1, [818].log_data[12].valid := 1, [818].log_data[13].valid := 1, [818].log_data[14].valid := 1, [818].log_data[15].valid := 1, [818].log_data[16].valid := 1, [818].log_data[17].valid := 1, [818].log_data[18].valid := 1, [818].log_data[19].valid := 1, [818].time.Year := 2023, [818].time.Month := 1, [818].time.Day := 12, [818].time.Hour := 12, [818].time.Minute := 34, [818].time.Second := 59, [819].log_data[0].min := 1.0, [819].log_data[0].max := 1.0, [819].log_data[0].total := 300.0, [819].log_data[0].time := 300.0, [819].log_data[0].minminute := 35, [819].log_data[0].maxminute := 35,
        [819].log_data[0].valid := 1, [819].log_data[1].valid := 1, [819].log_data[2].valid := 1, [819].log_data[3].valid := 1, [819].log_data[4].valid := 1, [819].log_data[5].valid := 1, [819].log_data[6].valid := 1, [819].log_data[7].valid := 1, [819].log_data[8].valid := 1, [819].log_data[9].valid := 1, [819].log_data[10].valid := 1, [819].log_data[11].valid := 1, [819].log_data[12].valid := 1, [819].log_data[13].valid := 1, [819].log_data[14].valid := 1, [819].log_data[15].valid := 1, [819].log_data[16].valid := 1, [819].log_data[17].valid := 1, [819].log_data[18].valid := 1, [819].log_data[19].valid := 1, [819].time.Year := 2023, [819].time.Month := 1, [819].time.Day := 12, [819].time.Hour := 12, [819].time.Minute := 39, [819].time.Second := 59, [820].log_data[0].min := 1.0, [820].log_data[0].max := 1.0, [820].log_data[0].total := 300.0, [820].log_data[0].time := 300.0, [820].log_data[0].minminute := 40, [820].log_data[0].maxminute := 40, [820].log_data[0].valid := 1, [820].log_data[1].valid := 1, [820].log_data[2].valid := 1, [820].log_data[3].valid := 1, [820].log_data[4].valid := 1, [820].log_data[5].valid := 1, [820].log_data[6].valid := 1, [820].log_data[7].valid := 1, [820].log_data[8].valid := 1, [820].log_data[9].valid := 1, [820].log_data[10].valid := 1, [820].log_data[11].valid := 1, [820].log_data[12].valid := 1, [820].log_data[13].valid := 1, [820].log_data[14].valid := 1, [820].log_data[15].valid := 1, [820].log_data[16].valid := 1, [820].log_data[17].valid := 1, [820].log_data[18].valid := 1, [820].log_data[19].valid := 1, [820].time.Year := 2023, [820].time.Month := 1, [820].time.Day := 12, [820].time.Hour := 12, [820].time.Minute := 44, [820].time.Second := 59, [821].log_data[0].min := 1.0, [821].log_data[0].max := 1.0,
        [821].log_data[0].total := 300.0, [821].log_data[0].time := 300.0, [821].log_data[0].minminute := 45, [821].log_data[0].maxminute := 45, [821].log_data[0].valid := 1, [821].log_data[1].valid := 1, [821].log_data[2].valid := 1, [821].log_data[3].valid := 1, [821].log_data[4].valid := 1, [821].log_data[5].valid := 1, [821].log_data[6].valid := 1, [821].log_data[7].valid := 1, [821].log_data[8].valid := 1, [821].log_data[9].valid := 1, [821].log_data[10].valid := 1, [821].log_data[11].valid := 1, [821].log_data[12].valid := 1, [821].log_data[13].valid := 1, [821].log_data[14].valid := 1, [821].log_data[15].valid := 1, [821].log_data[16].valid := 1, [821].log_data[17].valid := 1, [821].log_data[18].valid := 1, [821].log_data[19].valid := 1, [821].time.Year := 2023, [821].time.Month := 1, [821].time.Day := 12, [821].time.Hour := 12, [821].time.Minute := 49, [821].time.Second := 59, [822].log_data[0].min := 1.0, [822].log_data[0].max := 1.0, [822].log_data[0].total := 300.0, [822].log_data[0].time := 300.0, [822].log_data[0].minminute := 50, [822].log_data[0].maxminute := 50, [822].log_data[0].valid := 1, [822].log_data[1].valid := 1, [822].log_data[2].valid := 1, [822].log_data[3].valid := 1, [822].log_data[4].valid := 1, [822].log_data[5].valid := 1, [822].log_data[6].valid := 1, [822].log_data[7].valid := 1, [822].log_data[8].valid := 1, [822].log_data[9].valid := 1, [822].log_data[10].valid := 1, [822].log_data[11].valid := 1, [822].log_data[12].valid := 1, [822].log_data[13].valid := 1, [822].log_data[14].valid := 1, [822].log_data[15].valid := 1, [822].log_data[16].valid := 1, [822].log_data[17].valid := 1, [822].log_data[18].valid := 1, [822].log_data[19].valid := 1, [822].time.Year := 2023, [822].time.Month := 1, [822].time.Day := 12, [822].time.Hour := 12,
        [822].time.Minute := 54, [822].time.Second := 59, [823].log_data[0].min := 1.0, [823].log_data[0].max := 1.0, [823].log_data[0].total := 300.0, [823].log_data[0].time := 300.0, [823].log_data[0].minminute := 55, [823].log_data[0].maxminute := 55, [823].log_data[0].valid := 1, [823].log_data[1].valid := 1, [823].log_data[2].valid := 1, [823].log_data[3].valid := 1, [823].log_data[4].valid := 1, [823].log_data[5].valid := 1, [823].log_data[6].valid := 1, [823].log_data[7].valid := 1, [823].log_data[8].valid := 1, [823].log_data[9].valid := 1, [823].log_data[10].valid := 1, [823].log_data[11].valid := 1, [823].log_data[12].valid := 1, [823].log_data[13].valid := 1, [823].log_data[14].valid := 1, [823].log_data[15].valid := 1, [823].log_data[16].valid := 1, [823].log_data[17].valid := 1, [823].log_data[18].valid := 1, [823].log_data[19].valid := 1, [823].time.Year := 2023, [823].time.Month := 1, [823].time.Day := 12, [823].time.Hour := 12, [823].time.Minute := 59, [823].time.Second := 59, [824].log_data[0].min := 1.0, [824].log_data[0].max := 1.0, [824].log_data[0].total := 299.5, [824].log_data[0].time := 299.5, [824].log_data[0].valid := 1, [824].log_data[1].valid := 1, [824].log_data[2].valid := 1, [824].log_data[3].valid := 1, [824].log_data[4].valid := 1, [824].log_data[5].valid := 1, [824].log_data[6].valid := 1, [824].log_data[7].valid := 1, [824].log_data[8].valid := 1, [824].log_data[9].valid := 1, [824].log_data[10].valid := 1, [824].log_data[11].valid := 1, [824].log_data[12].valid := 1, [824].log_data[13].valid := 1, [824].log_data[14].valid := 1, [824].log_data[15].valid := 1, [824].log_data[16].valid := 1, [824].log_data[17].valid := 1, [824].log_data[18].valid := 1, [824].log_data[19].valid := 1, [824].time.Year := 2023, [824].time.Month := 1,
        [824].time.Day := 12, [824].time.Hour := 13, [824].time.Minute := 4, [824].time.Second := 59, [825].log_data[0].min := 1.0, [825].log_data[0].max := 1.0, [825].log_data[0].total := 300.0, [825].log_data[0].time := 300.0, [825].log_data[0].minminute := 5, [825].log_data[0].maxminute := 5, [825].log_data[0].valid := 1, [825].log_data[1].valid := 1, [825].log_data[2].valid := 1, [825].log_data[3].valid := 1, [825].log_data[4].valid := 1, [825].log_data[5].valid := 1, [825].log_data[6].valid := 1, [825].log_data[7].valid := 1, [825].log_data[8].valid := 1, [825].log_data[9].valid := 1, [825].log_data[10].valid := 1, [825].log_data[11].valid := 1, [825].log_data[12].valid := 1, [825].log_data[13].valid := 1, [825].log_data[14].valid := 1, [825].log_data[15].valid := 1, [825].log_data[16].valid := 1, [825].log_data[17].valid := 1, [825].log_data[18].valid := 1, [825].log_data[19].valid := 1, [825].time.Year := 2023, [825].time.Month := 1, [825].time.Day := 12, [825].time.Hour := 13, [825].time.Minute := 9, [825].time.Second := 59, [826].log_data[0].min := 1.0, [826].log_data[0].max := 1.0, [826].log_data[0].total := 300.0, [826].log_data[0].time := 300.0, [826].log_data[0].minminute := 10, [826].log_data[0].maxminute := 10, [826].log_data[0].valid := 1, [826].log_data[1].valid := 1, [826].log_data[2].valid := 1, [826].log_data[3].valid := 1, [826].log_data[4].valid := 1, [826].log_data[5].valid := 1, [826].log_data[6].valid := 1, [826].log_data[7].valid := 1, [826].log_data[8].valid := 1, [826].log_data[9].valid := 1, [826].log_data[10].valid := 1, [826].log_data[11].valid := 1, [826].log_data[12].valid := 1, [826].log_data[13].valid := 1, [826].log_data[14].valid := 1, [826].log_data[15].valid := 1, [826].log_data[16].valid := 1, [826].log_data[17].valid := 1,
        [826].log_data[18].valid := 1, [826].log_data[19].valid := 1, [826].time.Year := 2023, [826].time.Month := 1, [826].time.Day := 12, [826].time.Hour := 13, [826].time.Minute := 14, [826].time.Second := 59, [827].log_data[0].min := 1.0, [827].log_data[0].max := 1.0, [827].log_data[0].total := 300.0, [827].log_data[0].time := 300.0, [827].log_data[0].minminute := 15, [827].log_data[0].maxminute := 15, [827].log_data[0].valid := 1, [827].log_data[1].valid := 1, [827].log_data[2].valid := 1, [827].log_data[3].valid := 1, [827].log_data[4].valid := 1, [827].log_data[5].valid := 1, [827].log_data[6].valid := 1, [827].log_data[7].valid := 1, [827].log_data[8].valid := 1, [827].log_data[9].valid := 1, [827].log_data[10].valid := 1, [827].log_data[11].valid := 1, [827].log_data[12].valid := 1, [827].log_data[13].valid := 1, [827].log_data[14].valid := 1, [827].log_data[15].valid := 1, [827].log_data[16].valid := 1, [827].log_data[17].valid := 1, [827].log_data[18].valid := 1, [827].log_data[19].valid := 1, [827].time.Year := 2023, [827].time.Month := 1, [827].time.Day := 12, [827].time.Hour := 13, [827].time.Minute := 19, [827].time.Second := 59, [828].log_data[0].min := 1.0, [828].log_data[0].max := 1.0, [828].log_data[0].total := 300.0, [828].log_data[0].time := 300.0, [828].log_data[0].minminute := 20, [828].log_data[0].maxminute := 20, [828].log_data[0].valid := 1, [828].log_data[1].valid := 1, [828].log_data[2].valid := 1, [828].log_data[3].valid := 1, [828].log_data[4].valid := 1, [828].log_data[5].valid := 1, [828].log_data[6].valid := 1, [828].log_data[7].valid := 1, [828].log_data[8].valid := 1, [828].log_data[9].valid := 1, [828].log_data[10].valid := 1, [828].log_data[11].valid := 1, [828].log_data[12].valid := 1, [828].log_data[13].valid := 1,
        [828].log_data[14].valid := 1, [828].log_data[15].valid := 1, [828].log_data[16].valid := 1, [828].log_data[17].valid := 1, [828].log_data[18].valid := 1, [828].log_data[19].valid := 1, [828].time.Year := 2023, [828].time.Month := 1, [828].time.Day := 12, [828].time.Hour := 13, [828].time.Minute := 24, [828].time.Second := 59, [829].log_data[0].min := 1.0, [829].log_data[0].max := 1.0, [829].log_data[0].total := 300.0, [829].log_data[0].time := 300.0, [829].log_data[0].minminute := 25, [829].log_data[0].maxminute := 25, [829].log_data[0].valid := 1, [829].log_data[1].valid := 1, [829].log_data[2].valid := 1, [829].log_data[3].valid := 1, [829].log_data[4].valid := 1, [829].log_data[5].valid := 1, [829].log_data[6].valid := 1, [829].log_data[7].valid := 1, [829].log_data[8].valid := 1, [829].log_data[9].valid := 1, [829].log_data[10].valid := 1, [829].log_data[11].valid := 1, [829].log_data[12].valid := 1, [829].log_data[13].valid := 1, [829].log_data[14].valid := 1, [829].log_data[15].valid := 1, [829].log_data[16].valid := 1, [829].log_data[17].valid := 1, [829].log_data[18].valid := 1, [829].log_data[19].valid := 1, [829].time.Year := 2023, [829].time.Month := 1, [829].time.Day := 12, [829].time.Hour := 13, [829].time.Minute := 29, [829].time.Second := 59, [830].log_data[0].min := 1.0, [830].log_data[0].max := 1.0, [830].log_data[0].total := 300.0, [830].log_data[0].time := 300.0, [830].log_data[0].minminute := 30, [830].log_data[0].maxminute := 30, [830].log_data[0].valid := 1, [830].log_data[1].valid := 1, [830].log_data[2].valid := 1, [830].log_data[3].valid := 1, [830].log_data[4].valid := 1, [830].log_data[5].valid := 1, [830].log_data[6].valid := 1, [830].log_data[7].valid := 1, [830].log_data[8].valid := 1, [830].log_data[9].valid := 1,
        [830].log_data[10].valid := 1, [830].log_data[11].valid := 1, [830].log_data[12].valid := 1, [830].log_data[13].valid := 1, [830].log_data[14].valid := 1, [830].log_data[15].valid := 1, [830].log_data[16].valid := 1, [830].log_data[17].valid := 1, [830].log_data[18].valid := 1, [830].log_data[19].valid := 1, [830].time.Year := 2023, [830].time.Month := 1, [830].time.Day := 12, [830].time.Hour := 13, [830].time.Minute := 34, [830].time.Second := 59, [831].log_data[0].min := 1.0, [831].log_data[0].max := 1.0, [831].log_data[0].total := 300.0, [831].log_data[0].time := 300.0, [831].log_data[0].minminute := 35, [831].log_data[0].maxminute := 35, [831].log_data[0].valid := 1, [831].log_data[1].valid := 1, [831].log_data[2].valid := 1, [831].log_data[3].valid := 1, [831].log_data[4].valid := 1, [831].log_data[5].valid := 1, [831].log_data[6].valid := 1, [831].log_data[7].valid := 1, [831].log_data[8].valid := 1, [831].log_data[9].valid := 1, [831].log_data[10].valid := 1, [831].log_data[11].valid := 1, [831].log_data[12].valid := 1, [831].log_data[13].valid := 1, [831].log_data[14].valid := 1, [831].log_data[15].valid := 1, [831].log_data[16].valid := 1, [831].log_data[17].valid := 1, [831].log_data[18].valid := 1, [831].log_data[19].valid := 1, [831].time.Year := 2023, [831].time.Month := 1, [831].time.Day := 12, [831].time.Hour := 13, [831].time.Minute := 39, [831].time.Second := 59, [832].log_data[0].min := 1.0, [832].log_data[0].max := 1.0, [832].log_data[0].total := 300.0, [832].log_data[0].time := 300.0, [832].log_data[0].minminute := 40, [832].log_data[0].maxminute := 40, [832].log_data[0].valid := 1, [832].log_data[1].valid := 1, [832].log_data[2].valid := 1, [832].log_data[3].valid := 1, [832].log_data[4].valid := 1, [832].log_data[5].valid := 1,
        [832].log_data[6].valid := 1, [832].log_data[7].valid := 1, [832].log_data[8].valid := 1, [832].log_data[9].valid := 1, [832].log_data[10].valid := 1, [832].log_data[11].valid := 1, [832].log_data[12].valid := 1, [832].log_data[13].valid := 1, [832].log_data[14].valid := 1, [832].log_data[15].valid := 1, [832].log_data[16].valid := 1, [832].log_data[17].valid := 1, [832].log_data[18].valid := 1, [832].log_data[19].valid := 1, [832].time.Year := 2023, [832].time.Month := 1, [832].time.Day := 12, [832].time.Hour := 13, [832].time.Minute := 44, [832].time.Second := 59, [833].log_data[0].min := 1.0, [833].log_data[0].max := 1.0, [833].log_data[0].total := 300.0, [833].log_data[0].time := 300.0, [833].log_data[0].minminute := 45, [833].log_data[0].maxminute := 45, [833].log_data[0].valid := 1, [833].log_data[1].valid := 1, [833].log_data[2].valid := 1, [833].log_data[3].valid := 1, [833].log_data[4].valid := 1, [833].log_data[5].valid := 1, [833].log_data[6].valid := 1, [833].log_data[7].valid := 1, [833].log_data[8].valid := 1, [833].log_data[9].valid := 1, [833].log_data[10].valid := 1, [833].log_data[11].valid := 1, [833].log_data[12].valid := 1, [833].log_data[13].valid := 1, [833].log_data[14].valid := 1, [833].log_data[15].valid := 1, [833].log_data[16].valid := 1, [833].log_data[17].valid := 1, [833].log_data[18].valid := 1, [833].log_data[19].valid := 1, [833].time.Year := 2023, [833].time.Month := 1, [833].time.Day := 12, [833].time.Hour := 13, [833].time.Minute := 49, [833].time.Second := 59, [834].log_data[0].min := 1.0, [834].log_data[0].max := 1.0, [834].log_data[0].total := 300.0, [834].log_data[0].time := 300.0, [834].log_data[0].minminute := 50, [834].log_data[0].maxminute := 50, [834].log_data[0].valid := 1, [834].log_data[1].valid := 1,
        [834].log_data[2].valid := 1, [834].log_data[3].valid := 1, [834].log_data[4].valid := 1, [834].log_data[5].valid := 1, [834].log_data[6].valid := 1, [834].log_data[7].valid := 1, [834].log_data[8].valid := 1, [834].log_data[9].valid := 1, [834].log_data[10].valid := 1, [834].log_data[11].valid := 1, [834].log_data[12].valid := 1, [834].log_data[13].valid := 1, [834].log_data[14].valid := 1, [834].log_data[15].valid := 1, [834].log_data[16].valid := 1, [834].log_data[17].valid := 1, [834].log_data[18].valid := 1, [834].log_data[19].valid := 1, [834].time.Year := 2023, [834].time.Month := 1, [834].time.Day := 12, [834].time.Hour := 13, [834].time.Minute := 54, [834].time.Second := 59, [835].log_data[0].min := 1.0, [835].log_data[0].max := 1.0, [835].log_data[0].total := 300.0, [835].log_data[0].time := 300.0, [835].log_data[0].minminute := 55, [835].log_data[0].maxminute := 55, [835].log_data[0].valid := 1, [835].log_data[1].valid := 1, [835].log_data[2].valid := 1, [835].log_data[3].valid := 1, [835].log_data[4].valid := 1, [835].log_data[5].valid := 1, [835].log_data[6].valid := 1, [835].log_data[7].valid := 1, [835].log_data[8].valid := 1, [835].log_data[9].valid := 1, [835].log_data[10].valid := 1, [835].log_data[11].valid := 1, [835].log_data[12].valid := 1, [835].log_data[13].valid := 1, [835].log_data[14].valid := 1, [835].log_data[15].valid := 1, [835].log_data[16].valid := 1, [835].log_data[17].valid := 1, [835].log_data[18].valid := 1, [835].log_data[19].valid := 1, [835].time.Year := 2023, [835].time.Month := 1, [835].time.Day := 12, [835].time.Hour := 13, [835].time.Minute := 59, [835].time.Second := 59, [836].log_data[0].min := 1.0, [836].log_data[0].max := 1.0, [836].log_data[0].total := 300.0, [836].log_data[0].time := 300.0,
        [836].log_data[0].valid := 1, [836].log_data[1].valid := 1, [836].log_data[2].valid := 1, [836].log_data[3].valid := 1, [836].log_data[4].valid := 1, [836].log_data[5].valid := 1, [836].log_data[6].valid := 1, [836].log_data[7].valid := 1, [836].log_data[8].valid := 1, [836].log_data[9].valid := 1, [836].log_data[10].valid := 1, [836].log_data[11].valid := 1, [836].log_data[12].valid := 1, [836].log_data[13].valid := 1, [836].log_data[14].valid := 1, [836].log_data[15].valid := 1, [836].log_data[16].valid := 1, [836].log_data[17].valid := 1, [836].log_data[18].valid := 1, [836].log_data[19].valid := 1, [836].time.Year := 2023, [836].time.Month := 1, [836].time.Day := 12, [836].time.Hour := 14, [836].time.Minute := 4, [836].time.Second := 59, [837].log_data[0].min := 1.0, [837].log_data[0].max := 1.0, [837].log_data[0].total := 300.0, [837].log_data[0].time := 300.0, [837].log_data[0].minminute := 5, [837].log_data[0].maxminute := 5, [837].log_data[0].valid := 1, [837].log_data[1].valid := 1, [837].log_data[2].valid := 1, [837].log_data[3].valid := 1, [837].log_data[4].valid := 1, [837].log_data[5].valid := 1, [837].log_data[6].valid := 1, [837].log_data[7].valid := 1, [837].log_data[8].valid := 1, [837].log_data[9].valid := 1, [837].log_data[10].valid := 1, [837].log_data[11].valid := 1, [837].log_data[12].valid := 1, [837].log_data[13].valid := 1, [837].log_data[14].valid := 1, [837].log_data[15].valid := 1, [837].log_data[16].valid := 1, [837].log_data[17].valid := 1, [837].log_data[18].valid := 1, [837].log_data[19].valid := 1, [837].time.Year := 2023, [837].time.Month := 1, [837].time.Day := 12, [837].time.Hour := 14, [837].time.Minute := 9, [837].time.Second := 59, [838].log_data[0].min := 1.0, [838].log_data[0].max := 1.0,
        [838].log_data[0].total := 300.0, [838].log_data[0].time := 300.0, [838].log_data[0].minminute := 10, [838].log_data[0].maxminute := 10, [838].log_data[0].valid := 1, [838].log_data[1].valid := 1, [838].log_data[2].valid := 1, [838].log_data[3].valid := 1, [838].log_data[4].valid := 1, [838].log_data[5].valid := 1, [838].log_data[6].valid := 1, [838].log_data[7].valid := 1, [838].log_data[8].valid := 1, [838].log_data[9].valid := 1, [838].log_data[10].valid := 1, [838].log_data[11].valid := 1, [838].log_data[12].valid := 1, [838].log_data[13].valid := 1, [838].log_data[14].valid := 1, [838].log_data[15].valid := 1, [838].log_data[16].valid := 1, [838].log_data[17].valid := 1, [838].log_data[18].valid := 1, [838].log_data[19].valid := 1, [838].time.Year := 2023, [838].time.Month := 1, [838].time.Day := 12, [838].time.Hour := 14, [838].time.Minute := 14, [838].time.Second := 59, [839].log_data[0].min := 1.0, [839].log_data[0].max := 1.0, [839].log_data[0].total := 300.0, [839].log_data[0].time := 300.0, [839].log_data[0].minminute := 15, [839].log_data[0].maxminute := 15, [839].log_data[0].valid := 1, [839].log_data[1].valid := 1, [839].log_data[2].valid := 1, [839].log_data[3].valid := 1, [839].log_data[4].valid := 1, [839].log_data[5].valid := 1, [839].log_data[6].valid := 1, [839].log_data[7].valid := 1, [839].log_data[8].valid := 1, [839].log_data[9].valid := 1, [839].log_data[10].valid := 1, [839].log_data[11].valid := 1, [839].log_data[12].valid := 1, [839].log_data[13].valid := 1, [839].log_data[14].valid := 1, [839].log_data[15].valid := 1, [839].log_data[16].valid := 1, [839].log_data[17].valid := 1, [839].log_data[18].valid := 1, [839].log_data[19].valid := 1, [839].time.Year := 2023, [839].time.Month := 1, [839].time.Day := 12, [839].time.Hour := 14,
        [839].time.Minute := 19, [839].time.Second := 59, [840].log_data[0].min := 1.0, [840].log_data[0].max := 1.0, [840].log_data[0].total := 300.0, [840].log_data[0].time := 300.0, [840].log_data[0].minminute := 20, [840].log_data[0].maxminute := 20, [840].log_data[0].valid := 1, [840].log_data[1].valid := 1, [840].log_data[2].valid := 1, [840].log_data[3].valid := 1, [840].log_data[4].valid := 1, [840].log_data[5].valid := 1, [840].log_data[6].valid := 1, [840].log_data[7].valid := 1, [840].log_data[8].valid := 1, [840].log_data[9].valid := 1, [840].log_data[10].valid := 1, [840].log_data[11].valid := 1, [840].log_data[12].valid := 1, [840].log_data[13].valid := 1, [840].log_data[14].valid := 1, [840].log_data[15].valid := 1, [840].log_data[16].valid := 1, [840].log_data[17].valid := 1, [840].log_data[18].valid := 1, [840].log_data[19].valid := 1, [840].time.Year := 2023, [840].time.Month := 1, [840].time.Day := 12, [840].time.Hour := 14, [840].time.Minute := 24, [840].time.Second := 59, [841].log_data[0].min := 1.0, [841].log_data[0].max := 1.0, [841].log_data[0].total := 300.0, [841].log_data[0].time := 300.0, [841].log_data[0].minminute := 25, [841].log_data[0].maxminute := 25, [841].log_data[0].valid := 1, [841].log_data[1].valid := 1, [841].log_data[2].valid := 1, [841].log_data[3].valid := 1, [841].log_data[4].valid := 1, [841].log_data[5].valid := 1, [841].log_data[6].valid := 1, [841].log_data[7].valid := 1, [841].log_data[8].valid := 1, [841].log_data[9].valid := 1, [841].log_data[10].valid := 1, [841].log_data[11].valid := 1, [841].log_data[12].valid := 1, [841].log_data[13].valid := 1, [841].log_data[14].valid := 1, [841].log_data[15].valid := 1, [841].log_data[16].valid := 1, [841].log_data[17].valid := 1, [841].log_data[18].valid := 1, [841].log_data[19].valid := 1,
        [841].time.Year := 2023, [841].time.Month := 1, [841].time.Day := 12, [841].time.Hour := 14, [841].time.Minute := 29, [841].time.Second := 59, [842].log_data[0].min := 1.0, [842].log_data[0].max := 1.0, [842].log_data[0].total := 300.0, [842].log_data[0].time := 300.0, [842].log_data[0].minminute := 30, [842].log_data[0].maxminute := 30, [842].log_data[0].valid := 1, [842].log_data[1].valid := 1, [842].log_data[2].valid := 1, [842].log_data[3].valid := 1, [842].log_data[4].valid := 1, [842].log_data[5].valid := 1, [842].log_data[6].valid := 1, [842].log_data[7].valid := 1, [842].log_data[8].valid := 1, [842].log_data[9].valid := 1, [842].log_data[10].valid := 1, [842].log_data[11].valid := 1, [842].log_data[12].valid := 1, [842].log_data[13].valid := 1, [842].log_data[14].valid := 1, [842].log_data[15].valid := 1, [842].log_data[16].valid := 1, [842].log_data[17].valid := 1, [842].log_data[18].valid := 1, [842].log_data[19].valid := 1, [842].time.Year := 2023, [842].time.Month := 1, [842].time.Day := 12, [842].time.Hour := 14, [842].time.Minute := 34, [842].time.Second := 59, [843].log_data[0].min := 1.0, [843].log_data[0].max := 1.0, [843].log_data[0].total := 300.0, [843].log_data[0].time := 300.0, [843].log_data[0].minminute := 35, [843].log_data[0].maxminute := 35, [843].log_data[0].valid := 1, [843].log_data[1].valid := 1, [843].log_data[2].valid := 1, [843].log_data[3].valid := 1, [843].log_data[4].valid := 1, [843].log_data[5].valid := 1, [843].log_data[6].valid := 1, [843].log_data[7].valid := 1, [843].log_data[8].valid := 1, [843].log_data[9].valid := 1, [843].log_data[10].valid := 1, [843].log_data[11].valid := 1, [843].log_data[12].valid := 1, [843].log_data[13].valid := 1, [843].log_data[14].valid := 1, [843].log_data[15].valid := 1,
        [843].log_data[16].valid := 1, [843].log_data[17].valid := 1, [843].log_data[18].valid := 1, [843].log_data[19].valid := 1, [843].time.Year := 2023, [843].time.Month := 1, [843].time.Day := 12, [843].time.Hour := 14, [843].time.Minute := 39, [843].time.Second := 59, [844].log_data[0].min := 1.0, [844].log_data[0].max := 1.0, [844].log_data[0].total := 300.0, [844].log_data[0].time := 300.0, [844].log_data[0].minminute := 40, [844].log_data[0].maxminute := 40, [844].log_data[0].valid := 1, [844].log_data[1].valid := 1, [844].log_data[2].valid := 1, [844].log_data[3].valid := 1, [844].log_data[4].valid := 1, [844].log_data[5].valid := 1, [844].log_data[6].valid := 1, [844].log_data[7].valid := 1, [844].log_data[8].valid := 1, [844].log_data[9].valid := 1, [844].log_data[10].valid := 1, [844].log_data[11].valid := 1, [844].log_data[12].valid := 1, [844].log_data[13].valid := 1, [844].log_data[14].valid := 1, [844].log_data[15].valid := 1, [844].log_data[16].valid := 1, [844].log_data[17].valid := 1, [844].log_data[18].valid := 1, [844].log_data[19].valid := 1, [844].time.Year := 2023, [844].time.Month := 1, [844].time.Day := 12, [844].time.Hour := 14, [844].time.Minute := 44, [844].time.Second := 59, [845].log_data[0].min := 1.0, [845].log_data[0].max := 1.0, [845].log_data[0].total := 300.0, [845].log_data[0].time := 300.0, [845].log_data[0].minminute := 45, [845].log_data[0].maxminute := 45, [845].log_data[0].valid := 1, [845].log_data[1].valid := 1, [845].log_data[2].valid := 1, [845].log_data[3].valid := 1, [845].log_data[4].valid := 1, [845].log_data[5].valid := 1, [845].log_data[6].valid := 1, [845].log_data[7].valid := 1, [845].log_data[8].valid := 1, [845].log_data[9].valid := 1, [845].log_data[10].valid := 1, [845].log_data[11].valid := 1,
        [845].log_data[12].valid := 1, [845].log_data[13].valid := 1, [845].log_data[14].valid := 1, [845].log_data[15].valid := 1, [845].log_data[16].valid := 1, [845].log_data[17].valid := 1, [845].log_data[18].valid := 1, [845].log_data[19].valid := 1, [845].time.Year := 2023, [845].time.Month := 1, [845].time.Day := 12, [845].time.Hour := 14, [845].time.Minute := 49, [845].time.Second := 59, [846].log_data[0].min := 1.0, [846].log_data[0].max := 1.0, [846].log_data[0].total := 300.0, [846].log_data[0].time := 300.0, [846].log_data[0].minminute := 50, [846].log_data[0].maxminute := 50, [846].log_data[0].valid := 1, [846].log_data[1].valid := 1, [846].log_data[2].valid := 1, [846].log_data[3].valid := 1, [846].log_data[4].valid := 1, [846].log_data[5].valid := 1, [846].log_data[6].valid := 1, [846].log_data[7].valid := 1, [846].log_data[8].valid := 1, [846].log_data[9].valid := 1, [846].log_data[10].valid := 1, [846].log_data[11].valid := 1, [846].log_data[12].valid := 1, [846].log_data[13].valid := 1, [846].log_data[14].valid := 1, [846].log_data[15].valid := 1, [846].log_data[16].valid := 1, [846].log_data[17].valid := 1, [846].log_data[18].valid := 1, [846].log_data[19].valid := 1, [846].time.Year := 2023, [846].time.Month := 1, [846].time.Day := 12, [846].time.Hour := 14, [846].time.Minute := 54, [846].time.Second := 59, [847].log_data[0].min := 1.0, [847].log_data[0].max := 1.0, [847].log_data[0].total := 300.0, [847].log_data[0].time := 300.0, [847].log_data[0].minminute := 55, [847].log_data[0].maxminute := 55, [847].log_data[0].valid := 1, [847].log_data[1].valid := 1, [847].log_data[2].valid := 1, [847].log_data[3].valid := 1, [847].log_data[4].valid := 1, [847].log_data[5].valid := 1, [847].log_data[6].valid := 1, [847].log_data[7].valid := 1,
        [847].log_data[8].valid := 1, [847].log_data[9].valid := 1, [847].log_data[10].valid := 1, [847].log_data[11].valid := 1, [847].log_data[12].valid := 1, [847].log_data[13].valid := 1, [847].log_data[14].valid := 1, [847].log_data[15].valid := 1, [847].log_data[16].valid := 1, [847].log_data[17].valid := 1, [847].log_data[18].valid := 1, [847].log_data[19].valid := 1, [847].time.Year := 2023, [847].time.Month := 1, [847].time.Day := 12, [847].time.Hour := 14, [847].time.Minute := 59, [847].time.Second := 59, [848].log_data[0].min := 1.0, [848].log_data[0].max := 1.0, [848].log_data[0].total := 300.0, [848].log_data[0].time := 300.0, [848].log_data[0].valid := 1, [848].log_data[1].valid := 1, [848].log_data[2].valid := 1, [848].log_data[3].valid := 1, [848].log_data[4].valid := 1, [848].log_data[5].valid := 1, [848].log_data[6].valid := 1, [848].log_data[7].valid := 1, [848].log_data[8].valid := 1, [848].log_data[9].valid := 1, [848].log_data[10].valid := 1, [848].log_data[11].valid := 1, [848].log_data[12].valid := 1, [848].log_data[13].valid := 1, [848].log_data[14].valid := 1, [848].log_data[15].valid := 1, [848].log_data[16].valid := 1, [848].log_data[17].valid := 1, [848].log_data[18].valid := 1, [848].log_data[19].valid := 1, [848].time.Year := 2023, [848].time.Month := 1, [848].time.Day := 12, [848].time.Hour := 15, [848].time.Minute := 4, [848].time.Second := 59, [849].log_data[0].min := 1.0, [849].log_data[0].max := 1.0, [849].log_data[0].total := 300.0, [849].log_data[0].time := 300.0, [849].log_data[0].minminute := 5, [849].log_data[0].maxminute := 5, [849].log_data[0].valid := 1, [849].log_data[1].valid := 1, [849].log_data[2].valid := 1, [849].log_data[3].valid := 1, [849].log_data[4].valid := 1, [849].log_data[5].valid := 1,
        [849].log_data[6].valid := 1, [849].log_data[7].valid := 1, [849].log_data[8].valid := 1, [849].log_data[9].valid := 1, [849].log_data[10].valid := 1, [849].log_data[11].valid := 1, [849].log_data[12].valid := 1, [849].log_data[13].valid := 1, [849].log_data[14].valid := 1, [849].log_data[15].valid := 1, [849].log_data[16].valid := 1, [849].log_data[17].valid := 1, [849].log_data[18].valid := 1, [849].log_data[19].valid := 1, [849].time.Year := 2023, [849].time.Month := 1, [849].time.Day := 12, [849].time.Hour := 15, [849].time.Minute := 9, [849].time.Second := 59, [850].log_data[0].min := 1.0, [850].log_data[0].max := 1.0, [850].log_data[0].total := 300.0, [850].log_data[0].time := 300.0, [850].log_data[0].minminute := 10, [850].log_data[0].maxminute := 10, [850].log_data[0].valid := 1, [850].log_data[1].valid := 1, [850].log_data[2].valid := 1, [850].log_data[3].valid := 1, [850].log_data[4].valid := 1, [850].log_data[5].valid := 1, [850].log_data[6].valid := 1, [850].log_data[7].valid := 1, [850].log_data[8].valid := 1, [850].log_data[9].valid := 1, [850].log_data[10].valid := 1, [850].log_data[11].valid := 1, [850].log_data[12].valid := 1, [850].log_data[13].valid := 1, [850].log_data[14].valid := 1, [850].log_data[15].valid := 1, [850].log_data[16].valid := 1, [850].log_data[17].valid := 1, [850].log_data[18].valid := 1, [850].log_data[19].valid := 1, [850].time.Year := 2023, [850].time.Month := 1, [850].time.Day := 12, [850].time.Hour := 15, [850].time.Minute := 14, [850].time.Second := 59, [851].log_data[0].min := 1.0, [851].log_data[0].max := 1.0, [851].log_data[0].total := 300.0, [851].log_data[0].time := 300.0, [851].log_data[0].minminute := 15, [851].log_data[0].maxminute := 15, [851].log_data[0].valid := 1, [851].log_data[1].valid := 1,
        [851].log_data[2].valid := 1, [851].log_data[3].valid := 1, [851].log_data[4].valid := 1, [851].log_data[5].valid := 1, [851].log_data[6].valid := 1, [851].log_data[7].valid := 1, [851].log_data[8].valid := 1, [851].log_data[9].valid := 1, [851].log_data[10].valid := 1, [851].log_data[11].valid := 1, [851].log_data[12].valid := 1, [851].log_data[13].valid := 1, [851].log_data[14].valid := 1, [851].log_data[15].valid := 1, [851].log_data[16].valid := 1, [851].log_data[17].valid := 1, [851].log_data[18].valid := 1, [851].log_data[19].valid := 1, [851].time.Year := 2023, [851].time.Month := 1, [851].time.Day := 12, [851].time.Hour := 15, [851].time.Minute := 19, [851].time.Second := 59, [852].log_data[0].min := 1.0, [852].log_data[0].max := 1.0, [852].log_data[0].total := 300.0, [852].log_data[0].time := 300.0, [852].log_data[0].minminute := 20, [852].log_data[0].maxminute := 20, [852].log_data[0].valid := 1, [852].log_data[1].valid := 1, [852].log_data[2].valid := 1, [852].log_data[3].valid := 1, [852].log_data[4].valid := 1, [852].log_data[5].valid := 1, [852].log_data[6].valid := 1, [852].log_data[7].valid := 1, [852].log_data[8].valid := 1, [852].log_data[9].valid := 1, [852].log_data[10].valid := 1, [852].log_data[11].valid := 1, [852].log_data[12].valid := 1, [852].log_data[13].valid := 1, [852].log_data[14].valid := 1, [852].log_data[15].valid := 1, [852].log_data[16].valid := 1, [852].log_data[17].valid := 1, [852].log_data[18].valid := 1, [852].log_data[19].valid := 1, [852].time.Year := 2023, [852].time.Month := 1, [852].time.Day := 12, [852].time.Hour := 15, [852].time.Minute := 24, [852].time.Second := 59, [853].log_data[0].min := 1.0, [853].log_data[0].max := 1.0, [853].log_data[0].total := 300.0, [853].log_data[0].time := 300.0,
        [853].log_data[0].minminute := 25, [853].log_data[0].maxminute := 25, [853].log_data[0].valid := 1, [853].log_data[1].valid := 1, [853].log_data[2].valid := 1, [853].log_data[3].valid := 1, [853].log_data[4].valid := 1, [853].log_data[5].valid := 1, [853].log_data[6].valid := 1, [853].log_data[7].valid := 1, [853].log_data[8].valid := 1, [853].log_data[9].valid := 1, [853].log_data[10].valid := 1, [853].log_data[11].valid := 1, [853].log_data[12].valid := 1, [853].log_data[13].valid := 1, [853].log_data[14].valid := 1, [853].log_data[15].valid := 1, [853].log_data[16].valid := 1, [853].log_data[17].valid := 1, [853].log_data[18].valid := 1, [853].log_data[19].valid := 1, [853].time.Year := 2023, [853].time.Month := 1, [853].time.Day := 12, [853].time.Hour := 15, [853].time.Minute := 29, [853].time.Second := 59, [854].log_data[0].min := 1.0, [854].log_data[0].max := 1.0, [854].log_data[0].total := 300.0, [854].log_data[0].time := 300.0, [854].log_data[0].minminute := 30, [854].log_data[0].maxminute := 30, [854].log_data[0].valid := 1, [854].log_data[1].valid := 1, [854].log_data[2].valid := 1, [854].log_data[3].valid := 1, [854].log_data[4].valid := 1, [854].log_data[5].valid := 1, [854].log_data[6].valid := 1, [854].log_data[7].valid := 1, [854].log_data[8].valid := 1, [854].log_data[9].valid := 1, [854].log_data[10].valid := 1, [854].log_data[11].valid := 1, [854].log_data[12].valid := 1, [854].log_data[13].valid := 1, [854].log_data[14].valid := 1, [854].log_data[15].valid := 1, [854].log_data[16].valid := 1, [854].log_data[17].valid := 1, [854].log_data[18].valid := 1, [854].log_data[19].valid := 1, [854].time.Year := 2023, [854].time.Month := 1, [854].time.Day := 12, [854].time.Hour := 15, [854].time.Minute := 34, [854].time.Second := 59,
        [855].log_data[0].min := 1.0, [855].log_data[0].max := 1.0, [855].log_data[0].total := 300.0, [855].log_data[0].time := 300.0, [855].log_data[0].minminute := 35, [855].log_data[0].maxminute := 35, [855].log_data[0].valid := 1, [855].log_data[1].valid := 1, [855].log_data[2].valid := 1, [855].log_data[3].valid := 1, [855].log_data[4].valid := 1, [855].log_data[5].valid := 1, [855].log_data[6].valid := 1, [855].log_data[7].valid := 1, [855].log_data[8].valid := 1, [855].log_data[9].valid := 1, [855].log_data[10].valid := 1, [855].log_data[11].valid := 1, [855].log_data[12].valid := 1, [855].log_data[13].valid := 1, [855].log_data[14].valid := 1, [855].log_data[15].valid := 1, [855].log_data[16].valid := 1, [855].log_data[17].valid := 1, [855].log_data[18].valid := 1, [855].log_data[19].valid := 1, [855].time.Year := 2023, [855].time.Month := 1, [855].time.Day := 12, [855].time.Hour := 15, [855].time.Minute := 39, [855].time.Second := 59, [856].log_data[0].min := 1.0, [856].log_data[0].max := 1.0, [856].log_data[0].total := 300.0, [856].log_data[0].time := 300.0, [856].log_data[0].minminute := 40, [856].log_data[0].maxminute := 40, [856].log_data[0].valid := 1, [856].log_data[1].valid := 1, [856].log_data[2].valid := 1, [856].log_data[3].valid := 1, [856].log_data[4].valid := 1, [856].log_data[5].valid := 1, [856].log_data[6].valid := 1, [856].log_data[7].valid := 1, [856].log_data[8].valid := 1, [856].log_data[9].valid := 1, [856].log_data[10].valid := 1, [856].log_data[11].valid := 1, [856].log_data[12].valid := 1, [856].log_data[13].valid := 1, [856].log_data[14].valid := 1, [856].log_data[15].valid := 1, [856].log_data[16].valid := 1, [856].log_data[17].valid := 1, [856].log_data[18].valid := 1, [856].log_data[19].valid := 1, [856].time.Year := 2023, [856].time.Month := 1,
        [856].time.Day := 12, [856].time.Hour := 15, [856].time.Minute := 44, [856].time.Second := 59, [857].log_data[0].min := 1.0, [857].log_data[0].max := 1.0, [857].log_data[0].total := 300.0, [857].log_data[0].time := 300.0, [857].log_data[0].minminute := 45, [857].log_data[0].maxminute := 45, [857].log_data[0].valid := 1, [857].log_data[1].valid := 1, [857].log_data[2].valid := 1, [857].log_data[3].valid := 1, [857].log_data[4].valid := 1, [857].log_data[5].valid := 1, [857].log_data[6].valid := 1, [857].log_data[7].valid := 1, [857].log_data[8].valid := 1, [857].log_data[9].valid := 1, [857].log_data[10].valid := 1, [857].log_data[11].valid := 1, [857].log_data[12].valid := 1, [857].log_data[13].valid := 1, [857].log_data[14].valid := 1, [857].log_data[15].valid := 1, [857].log_data[16].valid := 1, [857].log_data[17].valid := 1, [857].log_data[18].valid := 1, [857].log_data[19].valid := 1, [857].time.Year := 2023, [857].time.Month := 1, [857].time.Day := 12, [857].time.Hour := 15, [857].time.Minute := 49, [857].time.Second := 59, [858].log_data[0].min := 1.0, [858].log_data[0].max := 1.0, [858].log_data[0].total := 300.0, [858].log_data[0].time := 300.0, [858].log_data[0].minminute := 50, [858].log_data[0].maxminute := 50, [858].log_data[0].valid := 1, [858].log_data[1].valid := 1, [858].log_data[2].valid := 1, [858].log_data[3].valid := 1, [858].log_data[4].valid := 1, [858].log_data[5].valid := 1, [858].log_data[6].valid := 1, [858].log_data[7].valid := 1, [858].log_data[8].valid := 1, [858].log_data[9].valid := 1, [858].log_data[10].valid := 1, [858].log_data[11].valid := 1, [858].log_data[12].valid := 1, [858].log_data[13].valid := 1, [858].log_data[14].valid := 1, [858].log_data[15].valid := 1, [858].log_data[16].valid := 1, [858].log_data[17].valid := 1,
        [858].log_data[18].valid := 1, [858].log_data[19].valid := 1, [858].time.Year := 2023, [858].time.Month := 1, [858].time.Day := 12, [858].time.Hour := 15, [858].time.Minute := 54, [858].time.Second := 59, [859].log_data[0].min := 1.0, [859].log_data[0].max := 1.0, [859].log_data[0].total := 300.0, [859].log_data[0].time := 300.0, [859].log_data[0].minminute := 55, [859].log_data[0].maxminute := 55, [859].log_data[0].valid := 1, [859].log_data[1].valid := 1, [859].log_data[2].valid := 1, [859].log_data[3].valid := 1, [859].log_data[4].valid := 1, [859].log_data[5].valid := 1, [859].log_data[6].valid := 1, [859].log_data[7].valid := 1, [859].log_data[8].valid := 1, [859].log_data[9].valid := 1, [859].log_data[10].valid := 1, [859].log_data[11].valid := 1, [859].log_data[12].valid := 1, [859].log_data[13].valid := 1, [859].log_data[14].valid := 1, [859].log_data[15].valid := 1, [859].log_data[16].valid := 1, [859].log_data[17].valid := 1, [859].log_data[18].valid := 1, [859].log_data[19].valid := 1, [859].time.Year := 2023, [859].time.Month := 1, [859].time.Day := 12, [859].time.Hour := 15, [859].time.Minute := 59, [859].time.Second := 59, [860].log_data[0].min := 1.0, [860].log_data[0].max := 1.0, [860].log_data[0].total := 300.0, [860].log_data[0].time := 300.0, [860].log_data[0].valid := 1, [860].log_data[1].valid := 1, [860].log_data[2].valid := 1, [860].log_data[3].valid := 1, [860].log_data[4].valid := 1, [860].log_data[5].valid := 1, [860].log_data[6].valid := 1, [860].log_data[7].valid := 1, [860].log_data[8].valid := 1, [860].log_data[9].valid := 1, [860].log_data[10].valid := 1, [860].log_data[11].valid := 1, [860].log_data[12].valid := 1, [860].log_data[13].valid := 1, [860].log_data[14].valid := 1, [860].log_data[15].valid := 1,
        [860].log_data[16].valid := 1, [860].log_data[17].valid := 1, [860].log_data[18].valid := 1, [860].log_data[19].valid := 1, [860].time.Year := 2023, [860].time.Month := 1, [860].time.Day := 12, [860].time.Hour := 16, [860].time.Minute := 4, [860].time.Second := 59, [861].log_data[0].min := 1.0, [861].log_data[0].max := 1.0, [861].log_data[0].total := 300.0, [861].log_data[0].time := 300.0, [861].log_data[0].minminute := 5, [861].log_data[0].maxminute := 5, [861].log_data[0].valid := 1, [861].log_data[1].valid := 1, [861].log_data[2].valid := 1, [861].log_data[3].valid := 1, [861].log_data[4].valid := 1, [861].log_data[5].valid := 1, [861].log_data[6].valid := 1, [861].log_data[7].valid := 1, [861].log_data[8].valid := 1, [861].log_data[9].valid := 1, [861].log_data[10].valid := 1, [861].log_data[11].valid := 1, [861].log_data[12].valid := 1, [861].log_data[13].valid := 1, [861].log_data[14].valid := 1, [861].log_data[15].valid := 1, [861].log_data[16].valid := 1, [861].log_data[17].valid := 1, [861].log_data[18].valid := 1, [861].log_data[19].valid := 1, [861].time.Year := 2023, [861].time.Month := 1, [861].time.Day := 12, [861].time.Hour := 16, [861].time.Minute := 9, [861].time.Second := 59, [862].log_data[0].min := 1.0, [862].log_data[0].max := 1.0, [862].log_data[0].total := 300.0, [862].log_data[0].time := 300.0, [862].log_data[0].minminute := 10, [862].log_data[0].maxminute := 10, [862].log_data[0].valid := 1, [862].log_data[1].valid := 1, [862].log_data[2].valid := 1, [862].log_data[3].valid := 1, [862].log_data[4].valid := 1, [862].log_data[5].valid := 1, [862].log_data[6].valid := 1, [862].log_data[7].valid := 1, [862].log_data[8].valid := 1, [862].log_data[9].valid := 1, [862].log_data[10].valid := 1, [862].log_data[11].valid := 1,
        [862].log_data[12].valid := 1, [862].log_data[13].valid := 1, [862].log_data[14].valid := 1, [862].log_data[15].valid := 1, [862].log_data[16].valid := 1, [862].log_data[17].valid := 1, [862].log_data[18].valid := 1, [862].log_data[19].valid := 1, [862].time.Year := 2023, [862].time.Month := 1, [862].time.Day := 12, [862].time.Hour := 16, [862].time.Minute := 14, [862].time.Second := 59, [863].log_data[0].min := 1.0, [863].log_data[0].max := 1.0, [863].log_data[0].total := 300.0, [863].log_data[0].time := 300.0, [863].log_data[0].minminute := 15, [863].log_data[0].maxminute := 15, [863].log_data[0].valid := 1, [863].log_data[1].valid := 1, [863].log_data[2].valid := 1, [863].log_data[3].valid := 1, [863].log_data[4].valid := 1, [863].log_data[5].valid := 1, [863].log_data[6].valid := 1, [863].log_data[7].valid := 1, [863].log_data[8].valid := 1, [863].log_data[9].valid := 1, [863].log_data[10].valid := 1, [863].log_data[11].valid := 1, [863].log_data[12].valid := 1, [863].log_data[13].valid := 1, [863].log_data[14].valid := 1, [863].log_data[15].valid := 1, [863].log_data[16].valid := 1, [863].log_data[17].valid := 1, [863].log_data[18].valid := 1, [863].log_data[19].valid := 1, [863].time.Year := 2023, [863].time.Month := 1, [863].time.Day := 12, [863].time.Hour := 16, [863].time.Minute := 19, [863].time.Second := 59, [864].log_data[0].min := 1.0, [864].log_data[0].max := 1.0, [864].log_data[0].total := 300.0, [864].log_data[0].time := 300.0, [864].log_data[0].minminute := 20, [864].log_data[0].maxminute := 20, [864].log_data[0].valid := 1, [864].log_data[1].valid := 1, [864].log_data[2].valid := 1, [864].log_data[3].valid := 1, [864].log_data[4].valid := 1, [864].log_data[5].valid := 1, [864].log_data[6].valid := 1, [864].log_data[7].valid := 1,
        [864].log_data[8].valid := 1, [864].log_data[9].valid := 1, [864].log_data[10].valid := 1, [864].log_data[11].valid := 1, [864].log_data[12].valid := 1, [864].log_data[13].valid := 1, [864].log_data[14].valid := 1, [864].log_data[15].valid := 1, [864].log_data[16].valid := 1, [864].log_data[17].valid := 1, [864].log_data[18].valid := 1, [864].log_data[19].valid := 1, [864].time.Year := 2023, [864].time.Month := 1, [864].time.Day := 12, [864].time.Hour := 16, [864].time.Minute := 24, [864].time.Second := 59, [865].log_data[0].min := 1.0, [865].log_data[0].max := 1.0, [865].log_data[0].total := 300.0, [865].log_data[0].time := 300.0, [865].log_data[0].minminute := 25, [865].log_data[0].maxminute := 25, [865].log_data[0].valid := 1, [865].log_data[1].valid := 1, [865].log_data[2].valid := 1, [865].log_data[3].valid := 1, [865].log_data[4].valid := 1, [865].log_data[5].valid := 1, [865].log_data[6].valid := 1, [865].log_data[7].valid := 1, [865].log_data[8].valid := 1, [865].log_data[9].valid := 1, [865].log_data[10].valid := 1, [865].log_data[11].valid := 1, [865].log_data[12].valid := 1, [865].log_data[13].valid := 1, [865].log_data[14].valid := 1, [865].log_data[15].valid := 1, [865].log_data[16].valid := 1, [865].log_data[17].valid := 1, [865].log_data[18].valid := 1, [865].log_data[19].valid := 1, [865].time.Year := 2023, [865].time.Month := 1, [865].time.Day := 12, [865].time.Hour := 16, [865].time.Minute := 29, [865].time.Second := 59, [866].log_data[0].min := 1.0, [866].log_data[0].max := 1.0, [866].log_data[0].total := 300.0, [866].log_data[0].time := 300.0, [866].log_data[0].minminute := 30, [866].log_data[0].maxminute := 30, [866].log_data[0].valid := 1, [866].log_data[1].valid := 1, [866].log_data[2].valid := 1, [866].log_data[3].valid := 1,
        [866].log_data[4].valid := 1, [866].log_data[5].valid := 1, [866].log_data[6].valid := 1, [866].log_data[7].valid := 1, [866].log_data[8].valid := 1, [866].log_data[9].valid := 1, [866].log_data[10].valid := 1, [866].log_data[11].valid := 1, [866].log_data[12].valid := 1, [866].log_data[13].valid := 1, [866].log_data[14].valid := 1, [866].log_data[15].valid := 1, [866].log_data[16].valid := 1, [866].log_data[17].valid := 1, [866].log_data[18].valid := 1, [866].log_data[19].valid := 1, [866].time.Year := 2023, [866].time.Month := 1, [866].time.Day := 12, [866].time.Hour := 16, [866].time.Minute := 34, [866].time.Second := 59, [867].log_data[0].min := 1.0, [867].log_data[0].max := 1.0, [867].log_data[0].total := 300.0, [867].log_data[0].time := 300.0, [867].log_data[0].minminute := 35, [867].log_data[0].maxminute := 35, [867].log_data[0].valid := 1, [867].log_data[1].valid := 1, [867].log_data[2].valid := 1, [867].log_data[3].valid := 1, [867].log_data[4].valid := 1, [867].log_data[5].valid := 1, [867].log_data[6].valid := 1, [867].log_data[7].valid := 1, [867].log_data[8].valid := 1, [867].log_data[9].valid := 1, [867].log_data[10].valid := 1, [867].log_data[11].valid := 1, [867].log_data[12].valid := 1, [867].log_data[13].valid := 1, [867].log_data[14].valid := 1, [867].log_data[15].valid := 1, [867].log_data[16].valid := 1, [867].log_data[17].valid := 1, [867].log_data[18].valid := 1, [867].log_data[19].valid := 1, [867].time.Year := 2023, [867].time.Month := 1, [867].time.Day := 12, [867].time.Hour := 16, [867].time.Minute := 39, [867].time.Second := 59, [868].log_data[0].min := 1.0, [868].log_data[0].max := 1.0, [868].log_data[0].total := 300.0, [868].log_data[0].time := 300.0, [868].log_data[0].minminute := 40, [868].log_data[0].maxminute := 40,
        [868].log_data[0].valid := 1, [868].log_data[1].valid := 1, [868].log_data[2].valid := 1, [868].log_data[3].valid := 1, [868].log_data[4].valid := 1, [868].log_data[5].valid := 1, [868].log_data[6].valid := 1, [868].log_data[7].valid := 1, [868].log_data[8].valid := 1, [868].log_data[9].valid := 1, [868].log_data[10].valid := 1, [868].log_data[11].valid := 1, [868].log_data[12].valid := 1, [868].log_data[13].valid := 1, [868].log_data[14].valid := 1, [868].log_data[15].valid := 1, [868].log_data[16].valid := 1, [868].log_data[17].valid := 1, [868].log_data[18].valid := 1, [868].log_data[19].valid := 1, [868].time.Year := 2023, [868].time.Month := 1, [868].time.Day := 12, [868].time.Hour := 16, [868].time.Minute := 44, [868].time.Second := 59, [869].log_data[0].min := 1.0, [869].log_data[0].max := 1.0, [869].log_data[0].total := 300.0, [869].log_data[0].time := 300.0, [869].log_data[0].minminute := 45, [869].log_data[0].maxminute := 45, [869].log_data[0].valid := 1, [869].log_data[1].valid := 1, [869].log_data[2].valid := 1, [869].log_data[3].valid := 1, [869].log_data[4].valid := 1, [869].log_data[5].valid := 1, [869].log_data[6].valid := 1, [869].log_data[7].valid := 1, [869].log_data[8].valid := 1, [869].log_data[9].valid := 1, [869].log_data[10].valid := 1, [869].log_data[11].valid := 1, [869].log_data[12].valid := 1, [869].log_data[13].valid := 1, [869].log_data[14].valid := 1, [869].log_data[15].valid := 1, [869].log_data[16].valid := 1, [869].log_data[17].valid := 1, [869].log_data[18].valid := 1, [869].log_data[19].valid := 1, [869].time.Year := 2023, [869].time.Month := 1, [869].time.Day := 12, [869].time.Hour := 16, [869].time.Minute := 49, [869].time.Second := 59, [870].log_data[0].min := 1.0, [870].log_data[0].max := 1.0,
        [870].log_data[0].total := 300.0, [870].log_data[0].time := 300.0, [870].log_data[0].minminute := 50, [870].log_data[0].maxminute := 50, [870].log_data[0].valid := 1, [870].log_data[1].valid := 1, [870].log_data[2].valid := 1, [870].log_data[3].valid := 1, [870].log_data[4].valid := 1, [870].log_data[5].valid := 1, [870].log_data[6].valid := 1, [870].log_data[7].valid := 1, [870].log_data[8].valid := 1, [870].log_data[9].valid := 1, [870].log_data[10].valid := 1, [870].log_data[11].valid := 1, [870].log_data[12].valid := 1, [870].log_data[13].valid := 1, [870].log_data[14].valid := 1, [870].log_data[15].valid := 1, [870].log_data[16].valid := 1, [870].log_data[17].valid := 1, [870].log_data[18].valid := 1, [870].log_data[19].valid := 1, [870].time.Year := 2023, [870].time.Month := 1, [870].time.Day := 12, [870].time.Hour := 16, [870].time.Minute := 54, [870].time.Second := 59, [871].log_data[0].min := 1.0, [871].log_data[0].max := 1.0, [871].log_data[0].total := 300.0, [871].log_data[0].time := 300.0, [871].log_data[0].minminute := 55, [871].log_data[0].maxminute := 55, [871].log_data[0].valid := 1, [871].log_data[1].valid := 1, [871].log_data[2].valid := 1, [871].log_data[3].valid := 1, [871].log_data[4].valid := 1, [871].log_data[5].valid := 1, [871].log_data[6].valid := 1, [871].log_data[7].valid := 1, [871].log_data[8].valid := 1, [871].log_data[9].valid := 1, [871].log_data[10].valid := 1, [871].log_data[11].valid := 1, [871].log_data[12].valid := 1, [871].log_data[13].valid := 1, [871].log_data[14].valid := 1, [871].log_data[15].valid := 1, [871].log_data[16].valid := 1, [871].log_data[17].valid := 1, [871].log_data[18].valid := 1, [871].log_data[19].valid := 1, [871].time.Year := 2023, [871].time.Month := 1, [871].time.Day := 12, [871].time.Hour := 16,
        [871].time.Minute := 59, [871].time.Second := 59, [872].log_data[0].min := 1.0, [872].log_data[0].max := 1.0, [872].log_data[0].total := 300.0, [872].log_data[0].time := 300.0, [872].log_data[0].valid := 1, [872].log_data[1].valid := 1, [872].log_data[2].valid := 1, [872].log_data[3].valid := 1, [872].log_data[4].valid := 1, [872].log_data[5].valid := 1, [872].log_data[6].valid := 1, [872].log_data[7].valid := 1, [872].log_data[8].valid := 1, [872].log_data[9].valid := 1, [872].log_data[10].valid := 1, [872].log_data[11].valid := 1, [872].log_data[12].valid := 1, [872].log_data[13].valid := 1, [872].log_data[14].valid := 1, [872].log_data[15].valid := 1, [872].log_data[16].valid := 1, [872].log_data[17].valid := 1, [872].log_data[18].valid := 1, [872].log_data[19].valid := 1, [872].time.Year := 2023, [872].time.Month := 1, [872].time.Day := 12, [872].time.Hour := 17, [872].time.Minute := 4, [872].time.Second := 59, [873].log_data[0].min := 1.0, [873].log_data[0].max := 1.0, [873].log_data[0].total := 300.0, [873].log_data[0].time := 300.0, [873].log_data[0].minminute := 5, [873].log_data[0].maxminute := 5, [873].log_data[0].valid := 1, [873].log_data[1].valid := 1, [873].log_data[2].valid := 1, [873].log_data[3].valid := 1, [873].log_data[4].valid := 1, [873].log_data[5].valid := 1, [873].log_data[6].valid := 1, [873].log_data[7].valid := 1, [873].log_data[8].valid := 1, [873].log_data[9].valid := 1, [873].log_data[10].valid := 1, [873].log_data[11].valid := 1, [873].log_data[12].valid := 1, [873].log_data[13].valid := 1, [873].log_data[14].valid := 1, [873].log_data[15].valid := 1, [873].log_data[16].valid := 1, [873].log_data[17].valid := 1, [873].log_data[18].valid := 1, [873].log_data[19].valid := 1, [873].time.Year := 2023, [873].time.Month := 1,
        [873].time.Day := 12, [873].time.Hour := 17, [873].time.Minute := 9, [873].time.Second := 59, [874].log_data[0].min := 1.0, [874].log_data[0].max := 1.0, [874].log_data[0].total := 300.0, [874].log_data[0].time := 300.0, [874].log_data[0].minminute := 10, [874].log_data[0].maxminute := 10, [874].log_data[0].valid := 1, [874].log_data[1].valid := 1, [874].log_data[2].valid := 1, [874].log_data[3].valid := 1, [874].log_data[4].valid := 1, [874].log_data[5].valid := 1, [874].log_data[6].valid := 1, [874].log_data[7].valid := 1, [874].log_data[8].valid := 1, [874].log_data[9].valid := 1, [874].log_data[10].valid := 1, [874].log_data[11].valid := 1, [874].log_data[12].valid := 1, [874].log_data[13].valid := 1, [874].log_data[14].valid := 1, [874].log_data[15].valid := 1, [874].log_data[16].valid := 1, [874].log_data[17].valid := 1, [874].log_data[18].valid := 1, [874].log_data[19].valid := 1, [874].time.Year := 2023, [874].time.Month := 1, [874].time.Day := 12, [874].time.Hour := 17, [874].time.Minute := 14, [874].time.Second := 59, [875].log_data[0].min := 1.0, [875].log_data[0].max := 1.0, [875].log_data[0].total := 300.0, [875].log_data[0].time := 300.0, [875].log_data[0].minminute := 15, [875].log_data[0].maxminute := 15, [875].log_data[0].valid := 1, [875].log_data[1].valid := 1, [875].log_data[2].valid := 1, [875].log_data[3].valid := 1, [875].log_data[4].valid := 1, [875].log_data[5].valid := 1, [875].log_data[6].valid := 1, [875].log_data[7].valid := 1, [875].log_data[8].valid := 1, [875].log_data[9].valid := 1, [875].log_data[10].valid := 1, [875].log_data[11].valid := 1, [875].log_data[12].valid := 1, [875].log_data[13].valid := 1, [875].log_data[14].valid := 1, [875].log_data[15].valid := 1, [875].log_data[16].valid := 1, [875].log_data[17].valid := 1,
        [875].log_data[18].valid := 1, [875].log_data[19].valid := 1, [875].time.Year := 2023, [875].time.Month := 1, [875].time.Day := 12, [875].time.Hour := 17, [875].time.Minute := 19, [875].time.Second := 59, [876].log_data[0].min := 1.0, [876].log_data[0].max := 1.0, [876].log_data[0].total := 300.0, [876].log_data[0].time := 300.0, [876].log_data[0].minminute := 20, [876].log_data[0].maxminute := 20, [876].log_data[0].valid := 1, [876].log_data[1].valid := 1, [876].log_data[2].valid := 1, [876].log_data[3].valid := 1, [876].log_data[4].valid := 1, [876].log_data[5].valid := 1, [876].log_data[6].valid := 1, [876].log_data[7].valid := 1, [876].log_data[8].valid := 1, [876].log_data[9].valid := 1, [876].log_data[10].valid := 1, [876].log_data[11].valid := 1, [876].log_data[12].valid := 1, [876].log_data[13].valid := 1, [876].log_data[14].valid := 1, [876].log_data[15].valid := 1, [876].log_data[16].valid := 1, [876].log_data[17].valid := 1, [876].log_data[18].valid := 1, [876].log_data[19].valid := 1, [876].time.Year := 2023, [876].time.Month := 1, [876].time.Day := 12, [876].time.Hour := 17, [876].time.Minute := 24, [876].time.Second := 59, [877].log_data[0].min := 1.0, [877].log_data[0].max := 1.0, [877].log_data[0].total := 300.0, [877].log_data[0].time := 300.0, [877].log_data[0].minminute := 25, [877].log_data[0].maxminute := 25, [877].log_data[0].valid := 1, [877].log_data[1].valid := 1, [877].log_data[2].valid := 1, [877].log_data[3].valid := 1, [877].log_data[4].valid := 1, [877].log_data[5].valid := 1, [877].log_data[6].valid := 1, [877].log_data[7].valid := 1, [877].log_data[8].valid := 1, [877].log_data[9].valid := 1, [877].log_data[10].valid := 1, [877].log_data[11].valid := 1, [877].log_data[12].valid := 1, [877].log_data[13].valid := 1,
        [877].log_data[14].valid := 1, [877].log_data[15].valid := 1, [877].log_data[16].valid := 1, [877].log_data[17].valid := 1, [877].log_data[18].valid := 1, [877].log_data[19].valid := 1, [877].time.Year := 2023, [877].time.Month := 1, [877].time.Day := 12, [877].time.Hour := 17, [877].time.Minute := 29, [877].time.Second := 59, [878].log_data[0].min := 1.0, [878].log_data[0].max := 1.0, [878].log_data[0].total := 300.0, [878].log_data[0].time := 300.0, [878].log_data[0].minminute := 30, [878].log_data[0].maxminute := 30, [878].log_data[0].valid := 1, [878].log_data[1].valid := 1, [878].log_data[2].valid := 1, [878].log_data[3].valid := 1, [878].log_data[4].valid := 1, [878].log_data[5].valid := 1, [878].log_data[6].valid := 1, [878].log_data[7].valid := 1, [878].log_data[8].valid := 1, [878].log_data[9].valid := 1, [878].log_data[10].valid := 1, [878].log_data[11].valid := 1, [878].log_data[12].valid := 1, [878].log_data[13].valid := 1, [878].log_data[14].valid := 1, [878].log_data[15].valid := 1, [878].log_data[16].valid := 1, [878].log_data[17].valid := 1, [878].log_data[18].valid := 1, [878].log_data[19].valid := 1, [878].time.Year := 2023, [878].time.Month := 1, [878].time.Day := 12, [878].time.Hour := 17, [878].time.Minute := 34, [878].time.Second := 59, [879].log_data[0].min := 1.0, [879].log_data[0].max := 1.0, [879].log_data[0].total := 300.0, [879].log_data[0].time := 300.0, [879].log_data[0].minminute := 35, [879].log_data[0].maxminute := 35, [879].log_data[0].valid := 1, [879].log_data[1].valid := 1, [879].log_data[2].valid := 1, [879].log_data[3].valid := 1, [879].log_data[4].valid := 1, [879].log_data[5].valid := 1, [879].log_data[6].valid := 1, [879].log_data[7].valid := 1, [879].log_data[8].valid := 1, [879].log_data[9].valid := 1,
        [879].log_data[10].valid := 1, [879].log_data[11].valid := 1, [879].log_data[12].valid := 1, [879].log_data[13].valid := 1, [879].log_data[14].valid := 1, [879].log_data[15].valid := 1, [879].log_data[16].valid := 1, [879].log_data[17].valid := 1, [879].log_data[18].valid := 1, [879].log_data[19].valid := 1, [879].time.Year := 2023, [879].time.Month := 1, [879].time.Day := 12, [879].time.Hour := 17, [879].time.Minute := 39, [879].time.Second := 59, [880].log_data[0].min := 1.0, [880].log_data[0].max := 1.0, [880].log_data[0].total := 300.0, [880].log_data[0].time := 300.0, [880].log_data[0].minminute := 40, [880].log_data[0].maxminute := 40, [880].log_data[0].valid := 1, [880].log_data[1].valid := 1, [880].log_data[2].valid := 1, [880].log_data[3].valid := 1, [880].log_data[4].valid := 1, [880].log_data[5].valid := 1, [880].log_data[6].valid := 1, [880].log_data[7].valid := 1, [880].log_data[8].valid := 1, [880].log_data[9].valid := 1, [880].log_data[10].valid := 1, [880].log_data[11].valid := 1, [880].log_data[12].valid := 1, [880].log_data[13].valid := 1, [880].log_data[14].valid := 1, [880].log_data[15].valid := 1, [880].log_data[16].valid := 1, [880].log_data[17].valid := 1, [880].log_data[18].valid := 1, [880].log_data[19].valid := 1, [880].time.Year := 2023, [880].time.Month := 1, [880].time.Day := 12, [880].time.Hour := 17, [880].time.Minute := 44, [880].time.Second := 59, [881].log_data[0].min := 1.0, [881].log_data[0].max := 1.0, [881].log_data[0].total := 300.0, [881].log_data[0].time := 300.0, [881].log_data[0].minminute := 45, [881].log_data[0].maxminute := 45, [881].log_data[0].valid := 1, [881].log_data[1].valid := 1, [881].log_data[2].valid := 1, [881].log_data[3].valid := 1, [881].log_data[4].valid := 1, [881].log_data[5].valid := 1,
        [881].log_data[6].valid := 1, [881].log_data[7].valid := 1, [881].log_data[8].valid := 1, [881].log_data[9].valid := 1, [881].log_data[10].valid := 1, [881].log_data[11].valid := 1, [881].log_data[12].valid := 1, [881].log_data[13].valid := 1, [881].log_data[14].valid := 1, [881].log_data[15].valid := 1, [881].log_data[16].valid := 1, [881].log_data[17].valid := 1, [881].log_data[18].valid := 1, [881].log_data[19].valid := 1, [881].time.Year := 2023, [881].time.Month := 1, [881].time.Day := 12, [881].time.Hour := 17, [881].time.Minute := 49, [881].time.Second := 59, [882].log_data[0].min := 1.0, [882].log_data[0].max := 1.0, [882].log_data[0].total := 300.0, [882].log_data[0].time := 300.0, [882].log_data[0].minminute := 50, [882].log_data[0].maxminute := 50, [882].log_data[0].valid := 1, [882].log_data[1].valid := 1, [882].log_data[2].valid := 1, [882].log_data[3].valid := 1, [882].log_data[4].valid := 1, [882].log_data[5].valid := 1, [882].log_data[6].valid := 1, [882].log_data[7].valid := 1, [882].log_data[8].valid := 1, [882].log_data[9].valid := 1, [882].log_data[10].valid := 1, [882].log_data[11].valid := 1, [882].log_data[12].valid := 1, [882].log_data[13].valid := 1, [882].log_data[14].valid := 1, [882].log_data[15].valid := 1, [882].log_data[16].valid := 1, [882].log_data[17].valid := 1, [882].log_data[18].valid := 1, [882].log_data[19].valid := 1, [882].time.Year := 2023, [882].time.Month := 1, [882].time.Day := 12, [882].time.Hour := 17, [882].time.Minute := 54, [882].time.Second := 59, [883].log_data[0].min := 1.0, [883].log_data[0].max := 1.0, [883].log_data[0].total := 300.0, [883].log_data[0].time := 300.0, [883].log_data[0].minminute := 55, [883].log_data[0].maxminute := 55, [883].log_data[0].valid := 1, [883].log_data[1].valid := 1,
        [883].log_data[2].valid := 1, [883].log_data[3].valid := 1, [883].log_data[4].valid := 1, [883].log_data[5].valid := 1, [883].log_data[6].valid := 1, [883].log_data[7].valid := 1, [883].log_data[8].valid := 1, [883].log_data[9].valid := 1, [883].log_data[10].valid := 1, [883].log_data[11].valid := 1, [883].log_data[12].valid := 1, [883].log_data[13].valid := 1, [883].log_data[14].valid := 1, [883].log_data[15].valid := 1, [883].log_data[16].valid := 1, [883].log_data[17].valid := 1, [883].log_data[18].valid := 1, [883].log_data[19].valid := 1, [883].time.Year := 2023, [883].time.Month := 1, [883].time.Day := 12, [883].time.Hour := 17, [883].time.Minute := 59, [883].time.Second := 59, [884].log_data[0].min := 1.0, [884].log_data[0].max := 1.0, [884].log_data[0].total := 300.0, [884].log_data[0].time := 300.0, [884].log_data[0].valid := 1, [884].log_data[1].valid := 1, [884].log_data[2].valid := 1, [884].log_data[3].valid := 1, [884].log_data[4].valid := 1, [884].log_data[5].valid := 1, [884].log_data[6].valid := 1, [884].log_data[7].valid := 1, [884].log_data[8].valid := 1, [884].log_data[9].valid := 1, [884].log_data[10].valid := 1, [884].log_data[11].valid := 1, [884].log_data[12].valid := 1, [884].log_data[13].valid := 1, [884].log_data[14].valid := 1, [884].log_data[15].valid := 1, [884].log_data[16].valid := 1, [884].log_data[17].valid := 1, [884].log_data[18].valid := 1, [884].log_data[19].valid := 1, [884].time.Year := 2023, [884].time.Month := 1, [884].time.Day := 12, [884].time.Hour := 18, [884].time.Minute := 4, [884].time.Second := 59, [885].log_data[0].min := 1.0, [885].log_data[0].max := 1.0, [885].log_data[0].total := 300.0, [885].log_data[0].time := 300.0, [885].log_data[0].minminute := 5, [885].log_data[0].maxminute := 5,
        [885].log_data[0].valid := 1, [885].log_data[1].valid := 1, [885].log_data[2].valid := 1, [885].log_data[3].valid := 1, [885].log_data[4].valid := 1, [885].log_data[5].valid := 1, [885].log_data[6].valid := 1, [885].log_data[7].valid := 1, [885].log_data[8].valid := 1, [885].log_data[9].valid := 1, [885].log_data[10].valid := 1, [885].log_data[11].valid := 1, [885].log_data[12].valid := 1, [885].log_data[13].valid := 1, [885].log_data[14].valid := 1, [885].log_data[15].valid := 1, [885].log_data[16].valid := 1, [885].log_data[17].valid := 1, [885].log_data[18].valid := 1, [885].log_data[19].valid := 1, [885].time.Year := 2023, [885].time.Month := 1, [885].time.Day := 12, [885].time.Hour := 18, [885].time.Minute := 9, [885].time.Second := 59, [886].log_data[0].min := 1.0, [886].log_data[0].max := 1.0, [886].log_data[0].total := 300.0, [886].log_data[0].time := 300.0, [886].log_data[0].minminute := 10, [886].log_data[0].maxminute := 10, [886].log_data[0].valid := 1, [886].log_data[1].valid := 1, [886].log_data[2].valid := 1, [886].log_data[3].valid := 1, [886].log_data[4].valid := 1, [886].log_data[5].valid := 1, [886].log_data[6].valid := 1, [886].log_data[7].valid := 1, [886].log_data[8].valid := 1, [886].log_data[9].valid := 1, [886].log_data[10].valid := 1, [886].log_data[11].valid := 1, [886].log_data[12].valid := 1, [886].log_data[13].valid := 1, [886].log_data[14].valid := 1, [886].log_data[15].valid := 1, [886].log_data[16].valid := 1, [886].log_data[17].valid := 1, [886].log_data[18].valid := 1, [886].log_data[19].valid := 1, [886].time.Year := 2023, [886].time.Month := 1, [886].time.Day := 12, [886].time.Hour := 18, [886].time.Minute := 14, [886].time.Second := 59, [887].log_data[0].min := 1.0, [887].log_data[0].max := 1.0,
        [887].log_data[0].total := 300.0, [887].log_data[0].time := 300.0, [887].log_data[0].minminute := 15, [887].log_data[0].maxminute := 15, [887].log_data[0].valid := 1, [887].log_data[1].valid := 1, [887].log_data[2].valid := 1, [887].log_data[3].valid := 1, [887].log_data[4].valid := 1, [887].log_data[5].valid := 1, [887].log_data[6].valid := 1, [887].log_data[7].valid := 1, [887].log_data[8].valid := 1, [887].log_data[9].valid := 1, [887].log_data[10].valid := 1, [887].log_data[11].valid := 1, [887].log_data[12].valid := 1, [887].log_data[13].valid := 1, [887].log_data[14].valid := 1, [887].log_data[15].valid := 1, [887].log_data[16].valid := 1, [887].log_data[17].valid := 1, [887].log_data[18].valid := 1, [887].log_data[19].valid := 1, [887].time.Year := 2023, [887].time.Month := 1, [887].time.Day := 12, [887].time.Hour := 18, [887].time.Minute := 19, [887].time.Second := 59, [888].log_data[0].min := 1.0, [888].log_data[0].max := 1.0, [888].log_data[0].total := 300.0, [888].log_data[0].time := 300.0, [888].log_data[0].minminute := 20, [888].log_data[0].maxminute := 20, [888].log_data[0].valid := 1, [888].log_data[1].valid := 1, [888].log_data[2].valid := 1, [888].log_data[3].valid := 1, [888].log_data[4].valid := 1, [888].log_data[5].valid := 1, [888].log_data[6].valid := 1, [888].log_data[7].valid := 1, [888].log_data[8].valid := 1, [888].log_data[9].valid := 1, [888].log_data[10].valid := 1, [888].log_data[11].valid := 1, [888].log_data[12].valid := 1, [888].log_data[13].valid := 1, [888].log_data[14].valid := 1, [888].log_data[15].valid := 1, [888].log_data[16].valid := 1, [888].log_data[17].valid := 1, [888].log_data[18].valid := 1, [888].log_data[19].valid := 1, [888].time.Year := 2023, [888].time.Month := 1, [888].time.Day := 12, [888].time.Hour := 18,
